KUKA KRL program: MyProgram_174().src

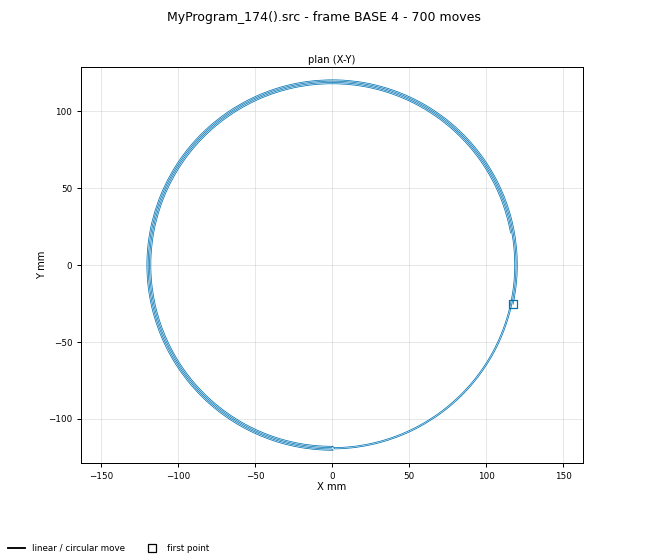
[picture p0: tool path of MyProgram_174().src in frame BASE 4, 700 of 700 moves have a stored position in this frame; points joined in program order, loops and branches not executed]
&ACCESS RVP
&REL 1
&PARAM TEMPLATE = C:\KRC\Roboter\Template\vorgabe
&PARAM EDITMASK = *
DEF MyProgram_174()
; ---- Setting reference (Base) ----
$BASE = BASE_DATA[4]

; --------------------------
; ---- Setting tool (TCP) ----
$TOOL = TOOL_DATA[3]
; --------------------------

$VEL.CP = VEL_APROX_PRINT
Startdeposition()
$VEL.CP = VEL_PRINT
LIN {X 117.5848,Y -25.4623,Z 129,A -15.6465,B 24.9508,C -1.6203,E1 25.1564,E2 461.721} C_DIS
LIN {X 118.3651,Y -21.5465,Z 129,A -14.0147,B 24.9512,C -1.6131,E1 25.1573,E2 460.1158} C_DIS
LIN {X 119.439,Y -14.4576,Z 129,A -10.3381,B 24.9498,C -1.6372,E1 25.1588,E2 456.4039} C_DIS
LIN {X 120.0869,Y -7.3562,Z 129,A -7.0535,B 24.9494,C -1.6427,E1 25.1596,E2 453.1258} C_DIS
LIN {X 120.304,Y -1.3301,Z 129,A -4.057,B 24.9485,C -1.6583,E1 25.1598,E2 450.1103} C_DIS
LIN {X 120.1794,Y 5.6204,Z 129,A -0.1852,B 24.946,C -1.6973,E1 25.1594,E2 446.1697} C_DIS
LIN {X 119.8532,Y 10.4886,Z 129,A 1.5179,B 24.9475,C -1.6737,E1 25.1591,E2 444.5324} C_DIS
LIN {X 119.0469,Y 17.3938,Z 129,A 5.2004,B 24.9457,C -1.7029,E1 25.1577,E2 440.8027} C_DIS
LIN {X 118.4357,Y 21.1537,Z 129,A 6.5409,B 24.9468,C -1.685,E1 25.1571,E2 439.5122} C_DIS
LIN {X 117.835,Y 24.2774,Z 129,A 8.2042,B 24.946,C -1.6972,E1 25.1562,E2 437.8299} C_DIS
LIN {X 116.908,Y 28.4078,Z 129,A 10.031,B 24.9462,C -1.6941,E1 25.155,E2 436.021} C_DIS
LIN {X 116.1551,Y 31.3444,Z 129,A 11.4464,B 24.946,C -1.6972,E1 25.154,E2 434.6064} C_DIS
LIN {X 115.3464,Y 34.2007,Z 129,A 12.8289,B 24.9458,C -1.7,E1 25.1529,E2 433.2252} C_DIS
LIN {X 114.4337,Y 37.1405,Z 129,A 14.334,B 24.9454,C -1.7065,E1 25.1517,E2 431.7135} C_DIS
LIN {X 113.2303,Y 40.6659,Z 129,A 16.6452,B 24.9434,C -1.7385,E1 25.1494,E2 429.3397} C_DIS
LIN {X 111.7337,Y 44.6139,Z 129,A 17.9875,B 24.9451,C -1.7113,E1 25.1482,E2 428.0691} C_DIS
LIN {X 110.031,Y 48.6627,Z 129,A 20.27,B 24.9441,C -1.7268,E1 25.1456,E2 425.7625} C_DIS
LIN {X 108.4702,Y 52.0451,Z 129,A 21.902,B 24.9442,C -1.7249,E1 25.1437,E2 424.1438} C_DIS
LIN {X 107.1163,Y 54.7776,Z 129,A 23.4021,B 24.9438,C -1.7314,E1 25.1418,E2 422.6363} C_DIS
LIN {X 105.3261,Y 58.1484,Z 129,A 25.0841,B 24.9439,C -1.7297,E1 25.1396,E2 420.9671} C_DIS
LIN {X 102.3478,Y 63.2435,Z 129,A 28.0641,B 24.9429,C -1.7456,E1 25.1353,E2 417.9649} C_DIS
LIN {X 100.5218,Y 66.105,Z 129,A 29.6094,B 24.9429,C -1.7464,E1 25.1329,E2 416.4254} C_DIS
LIN {X 98.1341,Y 69.6009,Z 129,A 31.5754,B 24.9427,C -1.7491,E1 25.1298,E2 414.4627} C_DIS
LIN {X 96.3458,Y 72.0557,Z 129,A 32.9323,B 24.9427,C -1.7484,E1 25.1276,E2 413.1141} C_DIS
LIN {X 94.6391,Y 74.2838,Z 129,A 34.2809,B 24.9425,C -1.7522,E1 25.1253,E2 411.7627} C_DIS
LIN {X 92.4033,Y 77.0464,Z 129,A 36.0716,B 24.9419,C -1.7611,E1 25.1221,E2 409.9593} C_DIS
LIN {X 89.7768,Y 80.0915,Z 129,A 37.9511,B 24.9417,C -1.7638,E1 25.1186,E2 408.0819} C_DIS
LIN {X 86.1601,Y 83.9723,Z 129,A 40.578,B 24.941,C -1.7743,E1 25.1136,E2 405.4416} C_DIS
LIN {X 83.2787,Y 86.8287,Z 129,A 43.2363,B 24.9383,C -1.8138,E1 25.1081,E2 402.701} C_DIS
LIN {X 79.152,Y 90.606,Z 129,A 45.0016,B 24.9409,C -1.7755,E1 25.1046,E2 401.0334} C_DIS
LIN {X 76.7994,Y 92.6085,Z 129,A 46.5139,B 24.9406,C -1.7803,E1 25.1013,E2 399.5155} C_DIS
LIN {X 73.8322,Y 94.9922,Z 129,A 48.3061,B 24.9404,C -1.7827,E1 25.0974,E2 397.7242} C_DIS
LIN {X 71.1983,Y 96.9809,Z 129,A 49.8066,B 24.9404,C -1.7821,E1 25.094,E2 396.2305} C_DIS
LIN {X 66.3731,Y 100.345,Z 129,A 52.681,B 24.9399,C -1.7903,E1 25.0874,E2 393.3466} C_DIS
LIN {X 63.7075,Y 102.058,Z 129,A 54.1758,B 24.9399,C -1.792,E1 25.0839,E2 391.8525} C_DIS
LIN {X 60.134,Y 104.2038,Z 129,A 56.1904,B 24.9395,C -1.7964,E1 25.079,E2 389.8338} C_DIS
LIN {X 56.8311,Y 106.0427,Z 129,A 58.0046,B 24.9393,C -1.7995,E1 25.0746,E2 388.0174} C_DIS
LIN {X 53.5539,Y 107.7333,Z 129,A 59.5541,B 24.9398,C -1.792,E1 25.0708,E2 386.4898} C_DIS
LIN {X 50.9117,Y 109.0069,Z 129,A 61.1282,B 24.9391,C -1.8021,E1 25.0667,E2 384.896} C_DIS
LIN {X 47.438,Y 110.5649,Z 129,A 62.9607,B 24.9389,C -1.8051,E1 25.0621,E2 383.0609} C_DIS
LIN {X 43.3807,Y 112.2186,Z 129,A 65.3004,B 24.938,C -1.8192,E1 25.0559,E2 380.6932} C_DIS
LIN {X 39.022,Y 113.8074,Z 129,A 67.1584,B 24.939,C -1.8046,E1 25.0511,E2 378.8734} C_DIS
LIN {X 35.8816,Y 114.8349,Z 129,A 68.9526,B 24.9382,C -1.8162,E1 25.0463,E2 377.055} C_DIS
LIN {X 31.5206,Y 116.1075,Z 129,A 70.8724,B 24.9388,C -1.8063,E1 25.0412,E2 375.1618} C_DIS
LIN {X 28.8672,Y 116.7959,Z 129,A 72.2811,B 24.9385,C -1.8119,E1 25.0373,E2 373.7419} C_DIS
LIN {X 25.2991,Y 117.6204,Z 129,A 74.3615,B 24.9373,C -1.8285,E1 25.0316,E2 371.625} C_DIS
LIN {X 21.8309,Y 118.3139,Z 129,A 75.7189,B 24.9383,C -1.814,E1 25.0279,E2 370.3036} C_DIS
LIN {X 18.5374,Y 118.8733,Z 129,A 77.239,B 24.9385,C -1.8112,E1 25.0238,E2 368.7915} C_DIS
LIN {X 15.7016,Y 119.2812,Z 129,A 78.6782,B 24.9383,C -1.815,E1 25.0198,E2 367.3445} C_DIS
LIN {X 9.3605,Y 119.9454,Z 129,A 81.6568,B 24.9384,C -1.8127,E1 25.0115,E2 364.3733} C_DIS
LIN {X 6.6678,Y 120.125,Z 129,A 83.2519,B 24.9374,C -1.827,E1 25.007,E2 362.745} C_DIS
LIN {X 2.0677,Y 120.2922,Z 129,A 85.7518,B 24.9365,C -1.8409,E1 24.9999,E2 360.2125} C_DIS
LIN {X -2.5546,Y 120.2833,Z 129,A 87.4564,B 24.9381,C -1.8174,E1 24.9953,E2 358.5634} C_DIS
LIN {X -9.7683,Y 119.9128,Z 129,A 90.5059,B 24.9394,C -1.7983,E1 24.9869,E2 355.5582} C_DIS
LIN {X -15.2296,Y 119.3423,Z 129,A 93.3875,B 24.9387,C -1.8089,E1 24.9789,E2 352.6498} C_DIS
LIN {X -18.4144,Y 118.8923,Z 129,A 95.5576,B 24.9368,C -1.8368,E1 24.9727,E2 350.4114} C_DIS
LIN {X -22.9909,Y 118.093,Z 129,A 97.1937,B 24.9387,C -1.8089,E1 24.9684,E2 348.84} C_DIS
LIN {X -26.6923,Y 117.3122,Z 129,A 98.9485,B 24.9389,C -1.8052,E1 24.9636,E2 347.0918} C_DIS
LIN {X -29.9813,Y 116.5144,Z 129,A 100.4878,B 24.9392,C -1.8004,E1 24.9594,E2 345.5618} C_DIS
LIN {X -33.4189,Y 115.5771,Z 129,A 102.3932,B 24.9387,C -1.8078,E1 24.9543,E2 343.6355} C_DIS
LIN {X -37.056,Y 114.461,Z 129,A 104.0991,B 24.9392,C -1.801,E1 24.9498,E2 341.9429} C_DIS
LIN {X -40.6481,Y 113.2369,Z 129,A 105.7919,B 24.9397,C -1.7936,E1 24.9453,E2 340.2643} C_DIS
LIN {X -46.0596,Y 111.1463,Z 129,A 108.7278,B 24.9394,C -1.7974,E1 24.9377,E2 337.313} C_DIS
LIN {X -49.0639,Y 109.8516,Z 129,A 110.2468,B 24.9397,C -1.7934,E1 24.9338,E2 335.8} C_DIS
LIN {X -54.1485,Y 107.4378,Z 129,A 112.984,B 24.9398,C -1.7916,E1 24.9269,E2 333.0599} C_DIS
LIN {X -57.1443,Y 105.8729,Z 129,A 114.6607,B 24.9398,C -1.7918,E1 24.9228,E2 331.3781} C_DIS
LIN {X -63.8759,Y 101.9528,Z 129,A 118.332,B 24.9404,C -1.7833,E1 24.914,E2 327.716} C_DIS
LIN {X -67.4437,Y 99.6284,Z 129,A 120.2451,B 24.941,C -1.7742,E1 24.9096,E2 325.818} C_DIS
LIN {X -71.7113,Y 96.6045,Z 129,A 122.8725,B 24.941,C -1.775,E1 24.9036,E2 323.1797} C_DIS
LIN {X -76.7717,Y 92.6316,Z 129,A 125.8608,B 24.9416,C -1.765,E1 24.8971,E2 320.2041} C_DIS
LIN {X -78.9489,Y 90.7833,Z 129,A 127.3315,B 24.9416,C -1.7667,E1 24.894,E2 318.7236} C_DIS
LIN {X -82.2494,Y 87.8041,Z 129,A 129.3861,B 24.942,C -1.759,E1 24.8898,E2 316.679} C_DIS
LIN {X -86.2573,Y 83.8715,Z 129,A 132.1268,B 24.9423,C -1.7553,E1 24.8843,E2 313.9355} C_DIS
LIN {X -89.1805,Y 80.7576,Z 129,A 134.1936,B 24.9425,C -1.7515,E1 24.8804,E2 311.8685} C_DIS
LIN {X -91.5631,Y 78.0428,Z 129,A 136.3235,B 24.9416,C -1.7649,E1 24.8765,E2 309.6971} C_DIS
LIN {X -94.1174,Y 74.9438,Z 129,A 137.6651,B 24.9436,C -1.735,E1 24.8743,E2 308.4205} C_DIS
LIN {X -97.8236,Y 70.0361,Z 129,A 141.1343,B 24.9426,C -1.7503,E1 24.8684,E2 304.8981} C_DIS
LIN {X -99.9834,Y 66.9195,Z 129,A 142.6448,B 24.9438,C -1.7324,E1 24.8661,E2 303.4226} C_DIS
LIN {X -102.0142,Y 63.7776,Z 129,A 144.293,B 24.9445,C -1.7216,E1 24.8637,E2 301.7919} C_DIS
LIN {X -103.3027,Y 61.671,Z 129,A 145.6708,B 24.9441,C -1.7268,E1 24.8617,E2 300.3945} C_DIS
LIN {X -106.9409,Y 55.1207,Z 129,A 148.9682,B 24.9455,C -1.7046,E1 24.8573,E2 297.1327} C_DIS
LIN {X -110.0031,Y 48.7267,Z 129,A 152.6095,B 24.9455,C -1.7056,E1 24.853,E2 293.4693} C_DIS
LIN {X -111.3647,Y 45.5238,Z 129,A 154.1469,B 24.9461,C -1.6953,E1 24.8513,E2 291.9477} C_DIS
LIN {X -112.6193,Y 42.3256,Z 129,A 157.0841,B 24.9428,C -1.7465,E1 24.8484,E2 288.872} C_DIS
LIN {X -115.0863,Y 35.0709,Z 129,A 159.0089,B 24.9483,C -1.6605,E1 24.8469,E2 287.1411} C_DIS
LIN {X -117.0482,Y 27.8334,Z 129,A 163.1341,B 24.9476,C -1.6724,E1 24.8439,E2 282.9634} C_DIS
LIN {X -117.7924,Y 24.4851,Z 129,A 164.7267,B 24.948,C -1.6654,E1 24.8429,E2 281.3782} C_DIS
LIN {X -118.3955,Y 21.3774,Z 129,A 166.2942,B 24.9482,C -1.6631,E1 24.8421,E2 279.8069} C_DIS
LIN {X -119.0397,Y 17.4443,Z 129,A 168.2482,B 24.9484,C -1.6593,E1 24.8413,E2 277.8504} C_DIS
LIN {X -119.4912,Y 14.0112,Z 129,A 169.8077,B 24.949,C -1.6501,E1 24.8407,E2 276.3035} C_DIS
LIN {X -119.8861,Y 10.1024,Z 129,A 171.7667,B 24.9491,C -1.6477,E1 24.8402,E2 274.3384} C_DIS
LIN {X -120.139,Y 6.4136,Z 129,A 173.4658,B 24.9496,C -1.6393,E1 24.84,E2 272.6491} C_DIS
LIN {X -120.28,Y 2.7339,Z 129,A 175.1714,B 24.9501,C -1.6315,E1 24.8398,E2 270.9518} C_DIS
LIN {X -120.3084,Y -0.6361,Z 129,A 176.8374,B 24.9503,C -1.6289,E1 24.8398,E2 269.2821} C_DIS
LIN {X -120.2335,Y -4.3356,Z 129,A 178.7511,B 24.9503,C -1.6296,E1 24.84,E2 267.3552} C_DIS
LIN {X -120.0348,Y -8.1312,Z 129,A -179.6085,B 24.951,C -1.6165,E1 24.8402,E2 265.7361} C_DIS
LIN {X -119.7828,Y -11.2509,Z 129,A -178.0156,B 24.951,C -1.6161,E1 24.8406,E2 264.1347} C_DIS
LIN {X -119.3925,Y -14.842,Z 129,A -176.2789,B 24.9514,C -1.6112,E1 24.8412,E2 262.3992} C_DIS
LIN {X -118.9209,Y -18.2295,Z 129,A -174.6385,B 24.9516,C -1.6065,E1 24.8418,E2 260.7603} C_DIS
LIN {X -118.257,Y -22.1389,Z 129,A -172.694,B 24.9519,C -1.6029,E1 24.8428,E2 258.8128} C_DIS
LIN {X -117.5326,Y -25.7013,Z 129,A -171.0443,B 24.9524,C -1.594,E1 24.8438,E2 257.1747} C_DIS
LIN {X -116.9844,Y -28.0949,Z 129,A -169.5097,B 24.9517,C -1.606,E1 24.8448,E2 255.6023} C_DIS
LIN {X -116.1801,Y -31.252,Z 129,A -167.2589,B 24.9501,C -1.6317,E1 24.8465,E2 253.2772} C_DIS
LIN {X -114.3114,Y -37.5184,Z 129,A -164.9234,B 24.9527,C -1.5882,E1 24.8484,E2 251.032} C_DIS
LIN {X -112.1931,Y -43.4456,Z 129,A -162.0631,B 24.9536,C -1.5733,E1 24.8512,E2 248.1912} C_DIS
LIN {X -110.8606,Y -46.7375,Z 129,A -160.4971,B 24.9542,C -1.5629,E1 24.8528,E2 246.6412} C_DIS
LIN {X -109.7148,Y -49.3674,Z 129,A -158.9868,B 24.9541,C -1.5652,E1 24.8546,E2 245.1172} C_DIS
LIN {X -107.9363,Y -53.1445,Z 129,A -157.0147,B 24.9545,C -1.5588,E1 24.8569,E2 243.1495} C_DIS
LIN {X -106.2522,Y -56.437,Z 129,A -155.3382,B 24.955,C -1.5502,E1 24.8591,E2 241.4846} C_DIS
LIN {X -103.1537,Y -61.9211,Z 129,A -152.1677,B 24.955,C -1.5494,E1 24.8635,E2 238.2994} C_DIS
LIN {X -101.2566,Y -64.9736,Z 129,A -150.6151,B 24.9557,C -1.538,E1 24.8658,E2 236.7662} C_DIS
LIN {X -98.4759,Y -69.1178,Z 129,A -148.0491,B 24.9556,C -1.5401,E1 24.8699,E2 234.1824} C_DIS
LIN {X -94.2815,Y -74.7362,Z 129,A -144.7252,B 24.9561,C -1.5312,E1 24.8755,E2 230.8638} C_DIS
LIN {X -91.7009,Y -77.881,Z 129,A -142.9284,B 24.9567,C -1.5204,E1 24.8787,E2 229.0844} C_DIS
LIN {X -86.961,Y -83.1415,Z 129,A -139.5195,B 24.957,C -1.5143,E1 24.8851,E2 225.6749} C_DIS
LIN {X -82.9842,Y -87.1125,Z 129,A -136.6202,B 24.9568,C -1.5185,E1 24.8909,E2 222.7537} C_DIS
LIN {X -79.8287,Y -90.012,Z 129,A -134.6188,B 24.9571,C -1.5126,E1 24.8951,E2 220.7582} C_DIS
LIN {X -76.4008,Y -92.9397,Z 129,A -132.5717,B 24.9576,C -1.504,E1 24.8994,E2 218.7237} C_DIS
LIN {X -73.5729,Y -95.1921,Z 129,A -131.0956,B 24.9584,C -1.49,E1 24.9026,E2 217.2755} C_DIS
LIN {X -70.5918,Y -97.4229,Z 129,A -128.601,B 24.9568,C -1.5191,E1 24.9084,E2 214.7028} C_DIS
LIN {X -67.4071,Y -99.6532,Z 129,A -127.2311,B 24.9582,C -1.4944,E1 24.9114,E2 213.3872} C_DIS
LIN {X -64.4112,Y -101.6176,Z 129,A -125.3419,B 24.9579,C -1.4999,E1 24.9159,E2 211.4787} C_DIS
LIN {X -61.2353,Y -103.5602,Z 129,A -123.7134,B 24.9584,C -1.4908,E1 24.9197,E2 209.867} C_DIS
LIN {X -57.9655,Y -105.4274,Z 129,A -121.8623,B 24.9584,C -1.4908,E1 24.9243,E2 208.0102} C_DIS
LIN {X -54.4907,Y -107.2628,Z 129,A -119.9679,B 24.9584,C -1.4895,E1 24.929,E2 206.114} C_DIS
LIN {X -50.8664,Y -109.028,Z 129,A -118.1583,B 24.9588,C -1.4822,E1 24.9335,E2 204.3171} C_DIS
LIN {X -46.2893,Y -111.0495,Z 129,A -115.4283,B 24.9581,C -1.4954,E1 24.9406,E2 201.5494} C_DIS
LIN {X -41.4285,Y -112.9522,Z 129,A -113.2356,B 24.959,C -1.4796,E1 24.9462,E2 199.3895} C_DIS
LIN {X -36.483,Y -114.6464,Z 129,A -110.7556,B 24.9591,C -1.4771,E1 24.9528,E2 196.9107} C_DIS
LIN {X -33.2199,Y -115.6335,Z 129,A -109.1067,B 24.9591,C -1.4771,E1 24.9572,E2 195.2591} C_DIS
LIN {X -30.3339,Y -116.4237,Z 129,A -107.609,B 24.959,C -1.4796,E1 24.9613,E2 193.7532} C_DIS
LIN {X -24.8979,Y -117.7076,Z 129,A -104.9009,B 24.959,C -1.4805,E1 24.9687,E2 191.0396} C_DIS
LIN {X -21.1668,Y -118.4333,Z 129,A -103.4454,B 24.9599,C -1.4635,E1 24.9726,E2 189.623} C_DIS
LIN {X -18.2676,Y -118.915,Z 129,A -101.9188,B 24.9596,C -1.4689,E1 24.9768,E2 188.082} C_DIS
LIN {X -11.8652,Y -119.7252,Z 129,A -98.4432,B 24.9586,C -1.4871,E1 24.9866,E2 184.561} C_DIS
LIN {X -6.1615,Y -120.153,Z 129,A -95.4276,B 24.9578,C -1.501,E1 24.9951,E2 181.5117} C_DIS
LIN {X -1.7022,Y -120.2989,Z 129,A -93.9382,B 24.9594,C -1.4714,E1 24.9991,E2 180.0922} C_DIS
LIN {X 0.8239,Y -120.3026,Z 129,A -91.9719,B 24.9574,C -1.5078,E1 25.0048,E2 178.0397} C_DIS
Enddeposition()
LIN {X 0.8239,Y -120.3026,Z 129,A -91.9719,B 24.9574,C -1.5078,E1 25.0048,E2 178.0397} C_DIS
Startdeposition()
$VEL.CP = VEL_PRINT
LIN {X -0.4367,Y -119.4615,Z 129,A -94.6116,B 24.9618,C -1.4278,E1 24.9969,E2 180.8689} C_DIS
LIN {X -4.7108,Y -119.3696,Z 129,A -96.1553,B 24.9606,C -1.4505,E1 24.9927,E2 182.3589} C_DIS
LIN {X -8.9928,Y -119.1241,Z 129,A -98.2312,B 24.9606,C -1.4496,E1 24.9869,E2 184.4378} C_DIS
LIN {X -12.4268,Y -118.8138,Z 129,A -100.1589,B 24.9613,C -1.4374,E1 24.9815,E2 186.3955} C_DIS
LIN {X -15.7199,Y -118.4237,Z 129,A -101.636,B 24.961,C -1.4428,E1 24.9774,E2 187.861} C_DIS
LIN {X -20.2124,Y -117.7407,Z 129,A -103.6777,B 24.9606,C -1.4497,E1 24.9718,E2 189.8882} C_DIS
LIN {X -23.8423,Y -117.0587,Z 129,A -105.3557,B 24.9604,C -1.4546,E1 24.9673,E2 191.5563} C_DIS
LIN {X -28.0159,Y -116.1308,Z 129,A -107.4362,B 24.9604,C -1.4543,E1 24.9616,E2 193.6404} C_DIS
LIN {X -31.5736,Y -115.2148,Z 129,A -109.1973,B 24.9604,C -1.4554,E1 24.9568,E2 195.4014} C_DIS
LIN {X -35.2602,Y -114.1397,Z 129,A -110.8974,B 24.9599,C -1.4631,E1 24.9523,E2 197.0862} C_DIS
LIN {X -37.9528,Y -113.2731,Z 129,A -112.4923,B 24.9604,C -1.4535,E1 24.948,E2 198.7067} C_DIS
LIN {X -41.8827,Y -111.8803,Z 129,A -114.5936,B 24.9606,C -1.4508,E1 24.9425,E2 200.8187} C_DIS
LIN {X -46.2868,Y -110.1303,Z 129,A -116.8437,B 24.9604,C -1.4542,E1 24.9367,E2 203.0659} C_DIS
LIN {X -50.2593,Y -108.3752,Z 129,A -118.7592,B 24.9599,C -1.4639,E1 24.9319,E2 204.9628} C_DIS
LIN {X -53.3538,Y -106.8861,Z 129,A -120.5285,B 24.96,C -1.4606,E1 24.9274,E2 206.7448} C_DIS
LIN {X -56.9088,Y -105.0359,Z 129,A -122.2931,B 24.9595,C -1.4701,E1 24.9231,E2 208.4917} C_DIS
LIN {X -59.5047,Y -103.5874,Z 129,A -123.7836,B 24.9595,C -1.4692,E1 24.9195,E2 209.9885} C_DIS
LIN {X -62.9285,Y -101.5447,Z 129,A -125.7339,B 24.9595,C -1.4704,E1 24.9148,E2 211.9421} C_DIS
LIN {X -65.9755,Y -99.5914,Z 129,A -127.414,B 24.9592,C -1.4756,E1 24.9109,E2 213.6152} C_DIS
LIN {X -71.648,Y -95.5914,Z 129,A -130.8507,B 24.9592,C -1.4766,E1 24.9031,E2 217.0614} C_DIS
LIN {X -75.1059,Y -92.8993,Z 129,A -132.9989,B 24.959,C -1.4785,E1 24.8983,E2 219.2131} C_DIS
LIN {X -78.417,Y -90.122,Z 129,A -134.955,B 24.9585,C -1.4876,E1 24.8942,E2 221.1552} C_DIS
LIN {X -80.9818,Y -87.8247,Z 129,A -136.5887,B 24.9583,C -1.4917,E1 24.8908,E2 222.7857} C_DIS
LIN {X -84.473,Y -84.4747,Z 129,A -139.0755,B 24.9584,C -1.4895,E1 24.8858,E2 225.2883} C_DIS
LIN {X -87.1368,Y -81.7212,Z 129,A -141.3008,B 24.9591,C -1.477,E1 24.8815,E2 227.5529} C_DIS
LIN {X -89.8475,Y -78.7312,Z 129,A -142.7343,B 24.9577,C -1.5029,E1 24.879,E2 228.9313} C_DIS
LIN {X -91.9677,Y -76.2437,Z 129,A -144.2811,B 24.9574,C -1.5075,E1 24.8762,E2 230.4743} C_DIS
LIN {X -93.5829,Y -74.2525,Z 129,A -146.3872,B 24.9593,C -1.4732,E1 24.8724,E2 232.6718} C_DIS
LIN {X -97.034,Y -69.6828,Z 129,A -148.1,B 24.9565,C -1.5239,E1 24.8697,E2 234.2722} C_DIS
LIN {X -99.5013,Y -66.1122,Z 129,A -150.4503,B 24.9568,C -1.5178,E1 24.866,E2 236.6488} C_DIS
LIN {X -101.3587,Y -63.2264,Z 129,A -152.0825,B 24.9566,C -1.5227,E1 24.8636,E2 238.2774} C_DIS
LIN {X -102.6529,Y -61.1037,Z 129,A -153.6613,B 24.9573,C -1.5096,E1 24.8613,E2 239.8957} C_DIS
LIN {X -104.4091,Y -58.0512,Z 129,A -155.2542,B 24.9568,C -1.5183,E1 24.8591,E2 241.4763} C_DIS
LIN {X -106.8872,Y -53.3516,Z 129,A -157.2967,B 24.9552,C -1.5468,E1 24.8566,E2 243.4617} C_DIS
LIN {X -107.7926,Y -51.4973,Z 129,A -158.616,B 24.9558,C -1.5356,E1 24.8549,E2 244.8147} C_DIS
LIN {X -109.4169,Y -47.9493,Z 129,A -160.3511,B 24.9552,C -1.5468,E1 24.8529,E2 246.5328} C_DIS
LIN {X -110.6429,Y -45.0478,Z 129,A -161.8964,B 24.955,C -1.5498,E1 24.8513,E2 248.0795} C_DIS
LIN {X -112.9279,Y -38.9721,Z 129,A -165.1325,B 24.9548,C -1.5539,E1 24.8482,E2 251.3242} C_DIS
LIN {X -114.0663,Y -35.497,Z 129,A -166.8077,B 24.9543,C -1.5626,E1 24.8467,E2 252.9882} C_DIS
LIN {X -115.2132,Y -31.5795,Z 129,A -169.4043,B 24.9555,C -1.542,E1 24.8448,E2 255.6491} C_DIS
LIN {X -116.3192,Y -27.2233,Z 129,A -170.9535,B 24.9536,C -1.5739,E1 24.8438,E2 257.1311} C_DIS
LIN {X -117.0179,Y -24.0408,Z 129,A -172.5595,B 24.9534,C -1.5771,E1 24.8428,E2 258.7391} C_DIS
LIN {X -117.7743,Y -20.0114,Z 129,A -174.5138,B 24.953,C -1.5838,E1 24.8419,E2 260.689} C_DIS
LIN {X -118.2819,Y -16.7494,Z 129,A -176.0889,B 24.9527,C -1.5892,E1 24.8412,E2 262.2606} C_DIS
LIN {X -118.7363,Y -13.1676,Z 129,A -177.979,B 24.9527,C -1.5881,E1 24.8406,E2 264.1645} C_DIS
LIN {X -119.0639,Y -9.7468,Z 129,A -179.5112,B 24.9521,C -1.5983,E1 24.8402,E2 265.6816} C_DIS
LIN {X -119.289,Y -6.4272,Z 129,A 178.8946,B 24.9518,C -1.6036,E1 24.84,E2 267.2728} C_DIS
LIN {X -119.4354,Y -2.54,Z 129,A 176.9999,B 24.9515,C -1.6084,E1 24.8398,E2 269.1673} C_DIS
LIN {X -119.459,Y 0.8647,Z 129,A 175.3431,B 24.9513,C -1.6128,E1 24.8398,E2 270.8238} C_DIS
LIN {X -119.3701,Y 4.7013,Z 129,A 173.4743,B 24.951,C -1.6176,E1 24.84,E2 272.6924} C_DIS
LIN {X -119.1844,Y 8.1378,Z 129,A 171.8667,B 24.9505,C -1.6248,E1 24.8402,E2 274.2924} C_DIS
LIN {X -118.8854,Y 11.7429,Z 129,A 169.9935,B 24.9505,C -1.6248,E1 24.8407,E2 276.1771} C_DIS
LIN {X -118.4752,Y 15.3227,Z 129,A 168.3806,B 24.9499,C -1.6352,E1 24.8412,E2 277.7747} C_DIS
LIN {X -117.9774,Y 18.7825,Z 129,A 166.5708,B 24.9499,C -1.6351,E1 24.842,E2 279.5955} C_DIS
LIN {X -117.3438,Y 22.3966,Z 129,A 164.9148,B 24.9493,C -1.6451,E1 24.8428,E2 281.2373} C_DIS
LIN {X -116.6098,Y 25.9531,Z 129,A 163.2229,B 24.9488,C -1.6528,E1 24.8438,E2 282.9209} C_DIS
LIN {X -115.0117,Y 32.3036,Z 129,A 159.9889,B 24.9484,C -1.659,E1 24.8461,E2 286.1591} C_DIS
LIN {X -113.8481,Y 36.1958,Z 129,A 157.1715,B 24.9503,C -1.6293,E1 24.8485,E2 289.0636} C_DIS
LIN {X -112.0446,Y 41.442,Z 129,A 155.2843,B 24.9478,C -1.6696,E1 24.8502,E2 290.8654} C_DIS
LIN {X -110.7115,Y 44.8791,Z 129,A 153.5762,B 24.9473,C -1.6776,E1 24.852,E2 292.5639} C_DIS
LIN {X -109.5996,Y 47.5304,Z 129,A 151.5129,B 24.9488,C -1.6534,E1 24.8544,E2 294.6961} C_DIS
LIN {X -107.6494,Y 51.7953,Z 129,A 149.89,B 24.9467,C -1.6862,E1 24.8562,E2 296.2497} C_DIS
LIN {X -105.9277,Y 55.2332,Z 129,A 147.9932,B 24.9465,C -1.6895,E1 24.8586,E2 298.1488} C_DIS
LIN {X -103.5203,Y 59.6214,Z 129,A 145.3426,B 24.9467,C -1.6862,E1 24.8623,E2 300.8213} C_DIS
LIN {X -101.0364,Y 63.7423,Z 129,A 143.2064,B 24.9458,C -1.7,E1 24.8654,E2 302.9355} C_DIS
LIN {X -98.2327,Y 67.982,Z 129,A 140.8781,B 24.9451,C -1.7115,E1 24.869,E2 305.248} C_DIS
LIN {X -96.3822,Y 70.5806,Z 129,A 138.9402,B 24.9459,C -1.6986,E1 24.8722,E2 307.2259} C_DIS
LIN {X -94.2532,Y 73.402,Z 129,A 137.6693,B 24.9445,C -1.721,E1 24.8743,E2 308.4496} C_DIS
LIN {X -91.033,Y 77.3574,Z 129,A 135.0344,B 24.9445,C -1.7195,E1 24.879,E2 311.1002} C_DIS
LIN {X -88.7077,Y 80.0143,Z 129,A 133.3566,B 24.9443,C -1.7245,E1 24.8821,E2 312.7736} C_DIS
LIN {X -85.5042,Y 83.4309,Z 129,A 130.8525,B 24.9446,C -1.7192,E1 24.887,E2 315.3011} C_DIS
LIN {X -81.3753,Y 87.4621,Z 129,A 128.3234,B 24.9435,C -1.7359,E1 24.892,E2 317.8009} C_DIS
LIN {X -78.2776,Y 90.2438,Z 129,A 126.2862,B 24.9433,C -1.7389,E1 24.8963,E2 319.8392} C_DIS
LIN {X -76.0959,Y 92.0906,Z 129,A 124.3675,B 24.9446,C -1.7188,E1 24.9006,E2 321.813} C_DIS
LIN {X -72.3363,Y 95.0744,Z 129,A 122.7641,B 24.9424,C -1.7533,E1 24.904,E2 323.3402} C_DIS
LIN {X -68.1659,Y 98.1048,Z 129,A 120.2546,B 24.9422,C -1.7568,E1 24.9097,E2 325.85} C_DIS
LIN {X -65.0999,Y 100.1679,Z 129,A 118.5149,B 24.9418,C -1.7617,E1 24.9137,E2 327.5839} C_DIS
LIN {X -60.6138,Y 102.9425,Z 129,A 115.3842,B 24.9432,C -1.7407,E1 24.9213,E2 330.774} C_DIS
LIN {X -57.049,Y 104.9599,Z 129,A 114.0051,B 24.9413,C -1.7692,E1 24.9245,E2 332.0893} C_DIS
LIN {X -51.6116,Y 107.7377,Z 129,A 110.9488,B 24.9413,C -1.7685,E1 24.9322,E2 335.1555} C_DIS
LIN {X -47.9493,Y 109.4169,Z 129,A 109.065,B 24.941,C -1.7735,E1 24.9369,E2 337.0318} C_DIS
LIN {X -42.8333,Y 111.5202,Z 129,A 106.5075,B 24.9405,C -1.7814,E1 24.9435,E2 339.5763} C_DIS
LIN {X -38.9198,Y 112.9462,Z 129,A 104.25,B 24.9411,C -1.7726,E1 24.9495,E2 341.8591} C_DIS
LIN {X -35.3618,Y 114.1083,Z 129,A 102.678,B 24.9403,C -1.7845,E1 24.9537,E2 343.4057} C_DIS
LIN {X -32.2489,Y 115.0273,Z 129,A 100.9668,B 24.9407,C -1.7794,E1 24.9583,E2 345.1317} C_DIS
LIN {X -28.3947,Y 116.0383,Z 129,A 99.1151,B 24.9404,C -1.7839,E1 24.9633,E2 346.9754} C_DIS
LIN {X -24.9598,Y 116.8264,Z 129,A 97.4056,B 24.9404,C -1.7846,E1 24.9679,E2 348.6854} C_DIS
LIN {X -20.1113,Y 117.7576,Z 129,A 95.052,B 24.9401,C -1.7871,E1 24.9744,E2 351.0356} C_DIS
LIN {X -17.052,Y 118.2389,Z 129,A 93.5048,B 24.9403,C -1.7854,E1 24.9787,E2 352.5883} C_DIS
LIN {X -11.5553,Y 118.9031,Z 129,A 90.8445,B 24.9402,C -1.7866,E1 24.9861,E2 355.2473} C_DIS
LIN {X -6.1538,Y 119.3041,Z 129,A 88.1952,B 24.9402,C -1.7854,E1 24.9934,E2 357.9004} C_DIS
LIN {X -2.1135,Y 119.4433,Z 129,A 86.0789,B 24.9407,C -1.7781,E1 24.9994,E2 360.0343} C_DIS
LIN {X 4.1595,Y 119.3905,Z 129,A 83.3177,B 24.94,C -1.7895,E1 25.007,E2 362.7679} C_DIS
LIN {X 7.8247,Y 119.2056,Z 129,A 81.5619,B 24.94,C -1.7897,E1 25.0119,E2 364.5226} C_DIS
LIN {X 12.7729,Y 118.7776,Z 129,A 79.0086,B 24.9405,C -1.7818,E1 25.0191,E2 367.0932} C_DIS
LIN {X 17.0048,Y 118.2456,Z 129,A 77.1012,B 24.9401,C -1.7875,E1 25.0243,E2 368.9854} C_DIS
LIN {X 20.9306,Y 117.6142,Z 129,A 75.2438,B 24.9401,C -1.7891,E1 25.0294,E2 370.8372} C_DIS
LIN {X 25.014,Y 116.8146,Z 129,A 73.2396,B 24.9401,C -1.7878,E1 25.0349,E2 372.842} C_DIS
LIN {X 28.3066,Y 116.0598,Z 129,A 71.6069,B 24.9401,C -1.7863,E1 25.0393,E2 374.4758} C_DIS
LIN {X 32.2713,Y 115.0209,Z 129,A 69.8444,B 24.9397,C -1.7943,E1 25.044,E2 376.2167} C_DIS
LIN {X 34.851,Y 114.2666,Z 129,A 68.2997,B 24.9405,C -1.7816,E1 25.0482,E2 377.7887} C_DIS
LIN {X 38.4073,Y 113.1198,Z 129,A 66.7299,B 24.9399,C -1.7903,E1 25.0523,E2 379.3348} C_DIS
LIN {X 41.7735,Y 111.9217,Z 129,A 64.8409,B 24.9406,C -1.7806,E1 25.0573,E2 381.2428} C_DIS
LIN {X 45.7752,Y 110.346,Z 129,A 62.7403,B 24.9408,C -1.7767,E1 25.0628,E2 383.3479} C_DIS
LIN {X 49.1876,Y 108.8657,Z 129,A 61.0523,B 24.9407,C -1.7792,E1 25.0671,E2 385.0259} C_DIS
LIN {X 52.7372,Y 107.1917,Z 129,A 59.179,B 24.9407,C -1.7773,E1 25.0718,E2 386.8989} C_DIS
LIN {X 55.6962,Y 105.6839,Z 129,A 57.6173,B 24.9408,C -1.7766,E1 25.0757,E2 388.4579} C_DIS
LIN {X 58.969,Y 103.8952,Z 129,A 55.7582,B 24.9412,C -1.7708,E1 25.0802,E2 390.3253} C_DIS
LIN {X 61.846,Y 102.207,Z 129,A 54.1757,B 24.9413,C -1.7692,E1 25.084,E2 391.9066} C_DIS
LIN {X 64.9082,Y 100.291,Z 129,A 52.429,B 24.9416,C -1.7658,E1 25.0881,E2 393.6558} C_DIS
LIN {X 67.515,Y 98.5561,Z 129,A 50.6854,B 24.9425,C -1.7519,E1 25.0922,E2 395.4261} C_DIS
LIN {X 71.5893,Y 95.6356,Z 129,A 48.5828,B 24.9418,C -1.7618,E1 25.0969,E2 397.4979} C_DIS
LIN {X 74.4478,Y 93.4286,Z 129,A 46.7658,B 24.9423,C -1.7546,E1 25.1009,E2 399.3252} C_DIS
LIN {X 77.4287,Y 90.9722,Z 129,A 45.0692,B 24.9421,C -1.7584,E1 25.1045,E2 401.0064} C_DIS
LIN {X 83.5476,Y 85.3889,Z 129,A 41.1962,B 24.9423,C -1.7548,E1 25.1125,E2 404.872} C_DIS
LIN {X 87.0944,Y 81.7663,Z 129,A 38.647,B 24.943,C -1.7438,E1 25.1174,E2 407.4362} C_DIS
LIN {X 89.7741,Y 78.8153,Z 129,A 36.7484,B 24.9433,C -1.7401,E1 25.1209,E2 409.3353} C_DIS
LIN {X 91.865,Y 76.3673,Z 129,A 35.3037,B 24.9432,C -1.7412,E1 25.1235,E2 410.7708} C_DIS
LIN {X 94.5274,Y 73.0462,Z 129,A 33.2033,B 24.9437,C -1.7334,E1 25.1272,E2 412.8797} C_DIS
LIN {X 96.6353,Y 70.2349,Z 129,A 31.3765,B 24.9444,C -1.7224,E1 25.1302,E2 414.7238} C_DIS
LIN {X 99.0786,Y 66.7433,Z 129,A 29.438,B 24.9444,C -1.7221,E1 25.1333,E2 416.6532} C_DIS
LIN {X 101.0866,Y 63.662,Z 129,A 27.7259,B 24.9446,C -1.72,E1 25.1359,E2 418.3619} C_DIS
LIN {X 102.526,Y 61.3185,Z 129,A 25.9649,B 24.9461,C -1.6952,E1 25.1385,E2 420.1723} C_DIS
LIN {X 104.3591,Y 58.1407,Z 129,A 24.6359,B 24.9451,C -1.711,E1 25.1402,E2 421.457} C_DIS
LIN {X 106.2039,Y 54.6995,Z 129,A 22.7666,B 24.9455,C -1.7059,E1 25.1427,E2 423.3285} C_DIS
LIN {X 107.6999,Y 51.6903,Z 129,A 21.2175,B 24.9455,C -1.7044,E1 25.1446,E2 424.8729} C_DIS
LIN {X 109.2243,Y 48.3912,Z 129,A 19.1639,B 24.9468,C -1.6843,E1 25.147,E2 426.9626} C_DIS
LIN {X 110.8373,Y 44.5701,Z 129,A 17.379,B 24.9466,C -1.6883,E1 25.1488,E2 428.7282} C_DIS
LIN {X 112.6997,Y 39.6223,Z 129,A 14.9328,B 24.9468,C -1.6851,E1 25.1512,E2 431.1685} C_DIS
LIN {X 113.9691,Y 35.8105,Z 129,A 13.037,B 24.9471,C -1.6807,E1 25.1528,E2 433.0638} C_DIS
LIN {X 114.8762,Y 32.7821,Z 129,A 11.5626,B 24.9472,C -1.6781,E1 25.154,E2 434.5361} C_DIS
LIN {X 115.6686,Y 29.8653,Z 129,A 10.0689,B 24.9476,C -1.6714,E1 25.155,E2 436.0369} C_DIS
LIN {X 116.4796,Y 26.5292,Z 129,A 8.4278,B 24.948,C -1.6665,E1 25.1561,E2 437.68} C_DIS
LIN {X 117.2536,Y 22.8656,Z 129,A 6.6651,B 24.9482,C -1.6624,E1 25.1571,E2 439.442} C_DIS
LIN {X 117.7305,Y 20.2738,Z 129,A 5.2526,B 24.9489,C -1.6512,E1 25.1578,E2 440.8728} C_DIS
LIN {X 118.587,Y 14.4419,Z 129,A 2.5537,B 24.9491,C -1.6483,E1 25.1588,E2 443.5625} C_DIS
LIN {X 118.9619,Y 10.9185,Z 129,A 1.0112,B 24.949,C -1.6505,E1 25.1592,E2 445.0908} C_DIS
LIN {X 119.2905,Y 6.4009,Z 129,A -1.5828,B 24.9506,C -1.6229,E1 25.1597,E2 447.7343} C_DIS
LIN {X 119.4287,Y 2.8979,Z 129,A -2.9779,B 24.9501,C -1.6313,E1 25.1597,E2 449.1014} C_DIS
LIN {X 119.4605,Y -0.6261,Z 129,A -4.5907,B 24.9502,C -1.6296,E1 25.1597,E2 450.7086} C_DIS
LIN {X 119.315,Y -5.9575,Z 129,A -7.1957,B 24.9509,C -1.6189,E1 25.1595,E2 453.3234} C_DIS
LIN {X 118.8893,Y -11.7027,Z 129,A -9.9649,B 24.9515,C -1.6095,E1 25.1589,E2 456.0982} C_DIS
LIN {X 118.428,Y -15.6866,Z 129,A -12.4004,B 24.9533,C -1.5783,E1 25.158,E2 458.5928} C_DIS
LIN {X 117.7147,Y -20.3678,Z 129,A -14.1101,B 24.9521,C -1.5982,E1 25.1572,E2 460.2457} C_DIS
LIN {X 117.0483,Y -23.8925,Z 129,A -15.6767,B 24.9521,C -1.6001,E1 25.1564,E2 461.7986} C_DIS
LIN {X 116.3764,Y -26.9756,Z 129,A -17.2446,B 24.9525,C -1.5925,E1 25.1554,E2 463.3753} C_DIS
LIN {X 115.4786,Y -30.5968,Z 129,A -19.0866,B 24.953,C -1.5842,E1 25.1541,E2 465.2263} C_DIS
LIN {X 114.4536,Y -34.2285,Z 129,A -20.8677,B 24.9532,C -1.5798,E1 25.1527,E2 467.0076} C_DIS
LIN {X 113.1972,Y -38.1778,Z 129,A -22.8663,B 24.9536,C -1.5729,E1 25.151,E2 469.011} C_DIS
LIN {X 111.7895,Y -42.1224,Z 129,A -24.7625,B 24.9536,C -1.5721,E1 25.1492,E2 470.8986} C_DIS
LIN {X 110.598,Y -45.1579,Z 129,A -26.3467,B 24.954,C -1.5662,E1 25.1475,E2 472.4879} C_DIS
LIN {X 109.0521,Y -48.774,Z 129,A -27.9812,B 24.9537,C -1.5727,E1 25.1458,E2 474.0982} C_DIS
LIN {X 107.215,Y -52.6902,Z 129,A -30.2935,B 24.9547,C -1.5547,E1 25.143,E2 476.4404} C_DIS
LIN {X 105.5693,Y -55.9138,Z 129,A -32.4251,B 24.9561,C -1.5303,E1 25.1401,E2 478.6182} C_DIS
LIN {X 103.7645,Y -59.1964,Z 129,A -33.8093,B 24.9553,C -1.545,E1 25.1383,E2 479.9607} C_DIS
LIN {X 100.9582,Y -63.8675,Z 129,A -36.4632,B 24.9558,C -1.5354,E1 25.1344,E2 482.6237} C_DIS
LIN {X 98.9604,Y -66.9178,Z 129,A -38.1024,B 24.9558,C -1.5358,E1 25.1319,E2 484.2539} C_DIS
LIN {X 97.5177,Y -69.0048,Z 129,A -40.0876,B 24.9581,C -1.4953,E1 25.1286,E2 486.3249} C_DIS
LIN {X 94.3866,Y -73.2289,Z 129,A -41.9461,B 24.9567,C -1.5203,E1 25.1255,E2 488.1157} C_DIS
LIN {X 91.496,Y -76.8113,Z 129,A -44.4171,B 24.9578,C -1.5017,E1 25.121,E2 490.6192} C_DIS
LIN {X 89.2285,Y -79.4326,Z 129,A -46.3174,B 24.9586,C -1.486,E1 25.1174,E2 492.548} C_DIS
LIN {X 86.0611,Y -82.8531,Z 129,A -47.8779,B 24.9571,C -1.5127,E1 25.1146,E2 494.0386} C_DIS
LIN {X 83.7201,Y -85.2185,Z 129,A -50.0233,B 24.9588,C -1.4824,E1 25.1102,E2 496.2465} C_DIS
LIN {X 80.6945,Y -88.0883,Z 129,A -51.8932,B 24.9588,C -1.4839,E1 25.1064,E2 498.1054} C_DIS
LIN {X 77.9118,Y -90.5607,Z 129,A -53.3345,B 24.9581,C -1.4962,E1 25.1034,E2 499.512} C_DIS
LIN {X 75.0923,Y -92.9103,Z 129,A -55.0065,B 24.9581,C -1.4965,E1 25.0998,E2 501.1769} C_DIS
LIN {X 70.9192,Y -96.1343,Z 129,A -57.7024,B 24.9588,C -1.483,E1 25.0938,E2 503.8948} C_DIS
LIN {X 67.2717,Y -98.7208,Z 129,A -59.7086,B 24.9587,C -1.4852,E1 25.0892,E2 505.889} C_DIS
LIN {X 60.5328,Y -102.9904,Z 129,A -63.0921,B 24.9579,C -1.4989,E1 25.0813,E2 509.2292} C_DIS
LIN {X 55.7994,Y -105.6295,Z 129,A -66.0452,B 24.9591,C -1.4773,E1 25.074,E2 512.2247} C_DIS
LIN {X 52.342,Y -107.3868,Z 129,A -68.4563,B 24.9607,C -1.4482,E1 25.0678,E2 514.6981} C_DIS
LIN {X 48.5308,Y -109.1617,Z 129,A -69.9596,B 24.9596,C -1.4692,E1 25.0641,E2 516.148} C_DIS
LIN {X 45.284,Y -110.5467,Z 129,A -71.6231,B 24.9596,C -1.4681,E1 25.0598,E2 517.8103} C_DIS
LIN {X 42.0707,Y -111.8091,Z 129,A -73.0979,B 24.9593,C -1.4744,E1 25.056,E2 519.2671} C_DIS
LIN {X 36.2985,Y -113.8149,Z 129,A -76.2641,B 24.9601,C -1.4595,E1 25.0476,E2 522.4622} C_DIS
LIN {X 32.6323,Y -114.9186,Z 129,A -78.0075,B 24.96,C -1.4618,E1 25.0429,E2 524.1972} C_DIS
LIN {X 28.99,Y -115.8931,Z 129,A -79.8847,B 24.9603,C -1.4566,E1 25.0378,E2 526.0838} C_DIS
LIN {X 25.4194,Y -116.7262,Z 129,A -81.5902,B 24.9603,C -1.4575,E1 25.0332,E2 527.785} C_DIS
LIN {X 20.9569,Y -117.6095,Z 129,A -83.9996,B 24.9609,C -1.4451,E1 25.0265,E2 530.2209} C_DIS
LIN {X 15.4106,Y -118.4638,Z 129,A -86.4146,B 24.9603,C -1.456,E1 25.0199,E2 532.6079} C_DIS
LIN {X 12.4982,Y -118.8063,Z 129,A -88.5374,B 24.9621,C -1.4223,E1 25.0138,E2 534.8091} C_DIS
LIN {X 7.5653,Y -119.2231,Z 129,A -90.14,B 24.9603,C -1.4565,E1 25.0096,E2 536.3299} C_DIS
LIN {X 1.7446,Y -119.45,Z 129,A -93.1245,B 24.9608,C -1.4468,E1 25.0012,E2 539.3367} C_DIS
LIN {X 1.7446,Y -119.45,Z 129,A -93.1245,B 24.9608,C -1.4468,E1 25.0012,E2 539.3367} C_DIS
Enddeposition()
LIN {X 0.8193,Y -118.6108,Z 129,A -93.4617,B 24.9597,C -1.4666,E1 25.0004,E2 539.627} C_DIS
Startdeposition()
$VEL.CP = VEL_PRINT
LIN {X 4.1826,Y -118.5414,Z 129,A -90.9638,B 24.9574,C -1.5072,E1 25.0076,E2 537.0335} C_DIS
LIN {X 7.3853,Y -118.3854,Z 129,A -89.5129,B 24.9577,C -1.5032,E1 25.0116,E2 535.5924} C_DIS
LIN {X 12.0231,Y -118.0035,Z 129,A -87.4079,B 24.958,C -1.4978,E1 25.0174,E2 533.5015} C_DIS
LIN {X 15.3204,Y -117.6204,Z 129,A -85.7262,B 24.9577,C -1.5025,E1 25.0221,E2 531.8101} C_DIS
LIN {X 18.6646,Y -117.1375,Z 129,A -83.7353,B 24.9567,C -1.5204,E1 25.0277,E2 529.7786} C_DIS
LIN {X 21.9525,Y -116.5658,Z 129,A -82.5812,B 24.9578,C -1.5003,E1 25.0308,E2 528.6734} C_DIS
LIN {X 24.4445,Y -116.0694,Z 129,A -81.2199,B 24.9574,C -1.5076,E1 25.0345,E2 527.2965} C_DIS
LIN {X 27.9179,Y -115.2818,Z 129,A -79.5222,B 24.9574,C -1.5083,E1 25.0391,E2 525.5996} C_DIS
LIN {X 30.9241,Y -114.5119,Z 129,A -78.0584,B 24.9574,C -1.5083,E1 25.0431,E2 524.1382} C_DIS
LIN {X 34.3845,Y -113.5228,Z 129,A -76.2046,B 24.957,C -1.5156,E1 25.0481,E2 522.2702} C_DIS
LIN {X 39.1081,Y -111.9815,Z 129,A -74.1386,B 24.9577,C -1.5029,E1 25.0535,E2 520.2383} C_DIS
LIN {X 42.0408,Y -110.9137,Z 129,A -72.4377,B 24.9571,C -1.514,E1 25.058,E2 518.5145} C_DIS
LIN {X 45.4847,Y -109.5482,Z 129,A -70.5036,B 24.9565,C -1.5235,E1 25.063,E2 516.5626} C_DIS
LIN {X 48.8644,Y -108.0813,Z 129,A -68.8477,B 24.9567,C -1.5203,E1 25.0672,E2 514.9181} C_DIS
LIN {X 52.6418,Y -106.2925,Z 129,A -66.8591,B 24.9566,C -1.5222,E1 25.0722,E2 512.9303} C_DIS
LIN {X 55.7558,Y -104.6941,Z 129,A -64.9869,B 24.9559,C -1.5338,E1 25.0769,E2 511.036} C_DIS
LIN {X 59.1528,Y -102.8116,Z 129,A -63.3298,B 24.9563,C -1.5267,E1 25.0809,E2 509.4006} C_DIS
LIN {X 62.1074,Y -101.0558,Z 129,A -61.3225,B 24.9552,C -1.5465,E1 25.0858,E2 507.3528} C_DIS
LIN {X 66.2431,Y -98.3931,Z 129,A -59.2375,B 24.9557,C -1.5372,E1 25.0906,E2 505.2965} C_DIS
LIN {X 69.1523,Y -96.3708,Z 129,A -57.5968,B 24.9557,C -1.5374,E1 25.0943,E2 503.6613} C_DIS
LIN {X 71.9229,Y -94.3224,Z 129,A -55.9409,B 24.9555,C -1.5405,E1 25.098,E2 502.0038} C_DIS
LIN {X 74.5558,Y -92.2536,Z 129,A -54.2824,B 24.9552,C -1.5461,E1 25.1016,E2 500.3383} C_DIS
LIN {X 77.3069,Y -89.962,Z 129,A -52.5023,B 24.9548,C -1.5525,E1 25.1054,E2 498.5501} C_DIS
LIN {X 80.6845,Y -86.9467,Z 129,A -50.274,B 24.9544,C -1.5597,E1 25.11,E2 496.3138} C_DIS
LIN {X 83.2266,Y -84.5141,Z 129,A -48.716,B 24.9546,C -1.557,E1 25.1131,E2 494.7687} C_DIS
LIN {X 85.5552,Y -82.1561,Z 129,A -47.0878,B 24.9543,C -1.5623,E1 25.1163,E2 493.1348} C_DIS
LIN {X 88.9632,Y -78.4547,Z 129,A -44.6644,B 24.9539,C -1.5682,E1 25.1209,E2 490.7082} C_DIS
LIN {X 90.9485,Y -76.1434,Z 129,A -43.183,B 24.9537,C -1.5726,E1 25.1235,E2 489.2233} C_DIS
LIN {X 93.1338,Y -73.4532,Z 129,A -41.5422,B 24.9535,C -1.5755,E1 25.1264,E2 487.5833} C_DIS
LIN {X 96.2908,Y -69.2644,Z 129,A -39.0311,B 24.9531,C -1.5814,E1 25.1306,E2 485.0704} C_DIS
LIN {X 98.3233,Y -66.3462,Z 129,A -37.3633,B 24.953,C -1.5838,E1 25.1332,E2 483.4051} C_DIS
LIN {X 100.3374,Y -63.2607,Z 129,A -35.4456,B 24.9523,C -1.5957,E1 25.1361,E2 481.4691} C_DIS
LIN {X 102.2328,Y -60.1479,Z 129,A -33.9059,B 24.9526,C -1.59,E1 25.1383,E2 479.9506} C_DIS
LIN {X 103.9616,Y -57.1109,Z 129,A -31.9908,B 24.9517,C -1.6061,E1 25.1409,E2 478.0075} C_DIS
LIN {X 105.9358,Y -53.3606,Z 129,A -29.8229,B 24.9509,C -1.6183,E1 25.1437,E2 475.8225} C_DIS
LIN {X 108.1415,Y -48.7307,Z 129,A -27.6686,B 24.9514,C -1.61,E1 25.1462,E2 473.6993} C_DIS
LIN {X 109.4996,Y -45.6,Z 129,A -26.0629,B 24.9512,C -1.613,E1 25.148,E2 472.0954} C_DIS
LIN {X 110.945,Y -41.958,Z 129,A -24.1517,B 24.9508,C -1.6198,E1 25.1499,E2 470.1787} C_DIS
LIN {X 112.2409,Y -38.36,Z 129,A -22.2224,B 24.9502,C -1.6297,E1 25.1517,E2 468.237} C_DIS
LIN {X 113.3953,Y -34.7979,Z 129,A -20.3909,B 24.9498,C -1.6366,E1 25.1532,E2 466.3997} C_DIS
LIN {X 114.498,Y -30.9754,Z 129,A -18.6016,B 24.9498,C -1.6362,E1 25.1546,E2 464.6214} C_DIS
LIN {X 115.2567,Y -28.0209,Z 129,A -17.1617,B 24.9496,C -1.6394,E1 25.1555,E2 463.1825} C_DIS
LIN {X 116.0286,Y -24.6385,Z 129,A -15.3733,B 24.949,C -1.6503,E1 25.1566,E2 461.3787} C_DIS
LIN {X 116.7673,Y -20.8492,Z 129,A -13.6384,B 24.949,C -1.65,E1 25.1575,E2 459.6546} C_DIS
LIN {X 117.4179,Y -16.8025,Z 129,A -11.6899,B 24.9487,C -1.6549,E1 25.1583,E2 457.706} C_DIS
LIN {X 117.8228,Y -13.6771,Z 129,A -10.1797,B 24.9484,C -1.6593,E1 25.1588,E2 456.1944} C_DIS
LIN {X 118.189,Y -10.0489,Z 129,A -8.2416,B 24.9475,C -1.6738,E1 25.1593,E2 454.2337} C_DIS
LIN {X 118.4784,Y -5.7015,Z 129,A -6.14,B 24.9471,C -1.6805,E1 25.1597,E2 452.1287} C_DIS
LIN {X 118.5914,Y -2.3172,Z 129,A -4.6768,B 24.9473,C -1.6774,E1 25.1597,E2 450.6815} C_DIS
LIN {X 118.6109,Y 0.8732,Z 129,A -3.105,B 24.9469,C -1.684,E1 25.1597,E2 449.1036} C_DIS
LIN {X 118.5085,Y 5.0003,Z 129,A -1.0941,B 24.9464,C -1.6913,E1 25.1596,E2 447.0874} C_DIS
LIN {X 118.29,Y 8.7862,Z 129,A 0.7853,B 24.9459,C -1.6996,E1 25.1592,E2 445.1996} C_DIS
LIN {X 117.9597,Y 12.4414,Z 129,A 2.3724,B 24.9461,C -1.6962,E1 25.1588,E2 443.6299} C_DIS
LIN {X 117.534,Y 15.9841,Z 129,A 4.2951,B 24.9451,C -1.7115,E1 25.1581,E2 441.6824} C_DIS
LIN {X 117.0009,Y 19.4949,Z 129,A 5.8353,B 24.9453,C -1.7084,E1 25.1574,E2 440.1586} C_DIS
LIN {X 116.3797,Y 22.9192,Z 129,A 7.5493,B 24.9449,C -1.7153,E1 25.1565,E2 438.4383} C_DIS
LIN {X 115.5597,Y 26.7438,Z 129,A 9.3285,B 24.9449,C -1.7159,E1 25.1554,E2 436.6681} C_DIS
LIN {X 114.8405,Y 29.6809,Z 129,A 10.8083,B 24.9445,C -1.7214,E1 25.1544,E2 435.1839} C_DIS
LIN {X 113.9226,Y 33.0369,Z 129,A 12.5511,B 24.9439,C -1.7296,E1 25.1531,E2 433.4318} C_DIS
LIN {X 112.8663,Y 36.4757,Z 129,A 14.2564,B 24.9437,C -1.7334,E1 25.1517,E2 431.7272} C_DIS
LIN {X 111.4795,Y 40.5167,Z 129,A 16.7246,B 24.942,C -1.7594,E1 25.1493,E2 429.2116} C_DIS
LIN {X 110.0926,Y 44.1503,Z 129,A 18.0886,B 24.9433,C -1.7398,E1 25.148,E2 427.9013} C_DIS
LIN {X 108.6572,Y 47.5701,Z 129,A 19.929,B 24.9428,C -1.7474,E1 25.1459,E2 426.053} C_DIS
LIN {X 107.0939,Y 50.9934,Z 129,A 21.7741,B 24.9423,C -1.7539,E1 25.1437,E2 424.2024} C_DIS
LIN {X 105.5543,Y 54.1071,Z 129,A 23.3719,B 24.9423,C -1.7548,E1 25.1417,E2 422.6111} C_DIS
LIN {X 103.8282,Y 57.3522,Z 129,A 25.3195,B 24.9414,C -1.7681,E1 25.1391,E2 420.6424} C_DIS
LIN {X 102.138,Y 60.3083,Z 129,A 26.7888,B 24.9417,C -1.7641,E1 25.1371,E2 419.1901} C_DIS
LIN {X 100.3541,Y 63.234,Z 129,A 28.4003,B 24.9415,C -1.7663,E1 25.1347,E2 417.5814} C_DIS
LIN {X 98.5407,Y 66.0251,Z 129,A 30.0725,B 24.941,C -1.7736,E1 25.1321,E2 415.9003} C_DIS
LIN {X 96.6369,Y 68.7793,Z 129,A 31.66,B 24.9409,C -1.7764,E1 25.1296,E2 414.3142} C_DIS
LIN {X 94.7585,Y 71.345,Z 129,A 33.1382,B 24.9408,C -1.7774,E1 25.1271,E2 412.8405} C_DIS
LIN {X 92.3701,Y 74.412,Z 129,A 35.0851,B 24.9403,C -1.7853,E1 25.1237,E2 410.8841} C_DIS
LIN {X 90.2547,Y 76.9634,Z 129,A 36.5773,B 24.9403,C -1.7839,E1 25.1211,E2 409.4021} C_DIS
LIN {X 88.2706,Y 79.2312,Z 129,A 38.0409,B 24.9401,C -1.7877,E1 25.1184,E2 407.9362} C_DIS
LIN {X 86.0277,Y 81.6628,Z 129,A 39.9087,B 24.939,C -1.8041,E1 25.1147,E2 406.0376} C_DIS
LIN {X 83.5209,Y 84.2234,Z 129,A 41.4033,B 24.9395,C -1.7966,E1 25.1118,E2 404.5672} C_DIS
LIN {X 81.1077,Y 86.5497,Z 129,A 43.5838,B 24.9374,C -1.8269,E1 25.1073,E2 402.3241} C_DIS
LIN {X 77.8802,Y 89.4649,Z 129,A 44.9924,B 24.9394,C -1.798,E1 25.1045,E2 400.9892} C_DIS
LIN {X 75.7462,Y 91.2786,Z 129,A 46.4064,B 24.939,C -1.8036,E1 25.1014,E2 399.5676} C_DIS
LIN {X 73.4219,Y 93.1585,Z 129,A 47.8617,B 24.9388,C -1.8068,E1 25.0982,E2 398.1101} C_DIS
LIN {X 70.374,Y 95.4825,Z 129,A 49.8528,B 24.9381,C -1.8167,E1 25.0937,E2 396.1026} C_DIS
LIN {X 67.6083,Y 97.4597,Z 129,A 51.4455,B 24.9381,C -1.8172,E1 25.0901,E2 394.5143} C_DIS
LIN {X 64.2388,Y 99.713,Z 129,A 53.3136,B 24.9381,C -1.8162,E1 25.0858,E2 392.6549} C_DIS
LIN {X 61.0355,Y 101.7073,Z 129,A 55.275,B 24.9375,C -1.8255,E1 25.0811,E2 390.6777} C_DIS
LIN {X 57.5551,Y 103.7149,Z 129,A 57.0063,B 24.938,C -1.8185,E1 25.0769,E2 388.9681} C_DIS
LIN {X 54.6923,Y 105.2542,Z 129,A 58.7457,B 24.9373,C -1.8285,E1 25.0726,E2 387.21} C_DIS
LIN {X 51.2843,Y 106.9541,Z 129,A 60.4465,B 24.9376,C -1.8243,E1 25.0683,E2 385.5235} C_DIS
LIN {X 48.1352,Y 108.4099,Z 129,A 62.2106,B 24.9372,C -1.8303,E1 25.0638,E2 383.7495} C_DIS
LIN {X 44.7569,Y 109.8458,Z 129,A 63.8847,B 24.9374,C -1.8277,E1 25.0595,E2 382.0856} C_DIS
LIN {X 41.4009,Y 111.156,Z 129,A 65.7293,B 24.9369,C -1.8342,E1 25.0547,E2 380.2296} C_DIS
LIN {X 37.7768,Y 112.4375,Z 129,A 67.514,B 24.9371,C -1.8325,E1 25.05,E2 378.4524} C_DIS
LIN {X 33.1074,Y 113.9017,Z 129,A 69.7671,B 24.9373,C -1.8292,E1 25.044,E2 376.2112} C_DIS
LIN {X 28.7014,Y 115.0907,Z 129,A 72.1636,B 24.9366,C -1.8394,E1 25.0375,E2 373.7941} C_DIS
LIN {X 25.2542,Y 115.8943,Z 129,A 73.8124,B 24.9367,C -1.8375,E1 25.033,E2 372.152} C_DIS
LIN {X 21.9828,Y 116.56,Z 129,A 75.3464,B 24.9369,C -1.8346,E1 25.0288,E2 370.6267} C_DIS
LIN {X 18.5434,Y 117.1562,Z 129,A 77.0863,B 24.9367,C -1.8377,E1 25.024,E2 368.8814} C_DIS
LIN {X 15.129,Y 117.6452,Z 129,A 78.7105,B 24.9368,C -1.8362,E1 25.0195,E2 367.2621} C_DIS
LIN {X 11.8301,Y 118.0237,Z 129,A 80.2797,B 24.9368,C -1.8348,E1 25.0152,E2 365.6972} C_DIS
LIN {X 9.2808,Y 118.2504,Z 129,A 81.6183,B 24.9366,C -1.8396,E1 25.0114,E2 364.3481} C_DIS
LIN {X 4.9925,Y 118.5089,Z 129,A 83.6071,B 24.9368,C -1.8356,E1 25.0059,E2 362.3693} C_DIS
LIN {X 1.9365,Y 118.5984,Z 129,A 85.2138,B 24.9365,C -1.8413,E1 25.0014,E2 360.7495} C_DIS
LIN {X -2.2681,Y 118.5923,Z 129,A 87.142,B 24.9368,C -1.8362,E1 24.996,E2 358.8333} C_DIS
LIN {X -5.6323,Y 118.4814,Z 129,A 88.8902,B 24.9365,C -1.8411,E1 24.9911,E2 357.0731} C_DIS
LIN {X -10.0384,Y 118.1899,Z 129,A 91.0271,B 24.9365,C -1.8403,E1 24.9852,E2 354.9371} C_DIS
LIN {X -14.7549,Y 117.6937,Z 129,A 93.2402,B 24.9368,C -1.8356,E1 24.9791,E2 352.7338} C_DIS
LIN {X -18.0836,Y 117.2273,Z 129,A 94.9023,B 24.9368,C -1.8362,E1 24.9745,E2 351.0689} C_DIS
LIN {X -21.8698,Y 116.5817,Z 129,A 96.8236,B 24.9367,C -1.8377,E1 24.9692,E2 349.1421} C_DIS
LIN {X -25.8853,Y 115.7567,Z 129,A 98.793,B 24.9369,C -1.8355,E1 24.9638,E2 347.1756} C_DIS
LIN {X -29.6654,Y 114.8445,Z 129,A 100.5525,B 24.9373,C -1.8284,E1 24.9591,E2 345.4304} C_DIS
LIN {X -33.0909,Y 113.9066,Z 129,A 102.4912,B 24.9368,C -1.8364,E1 24.9538,E2 343.4697} C_DIS
LIN {X -36.6981,Y 112.7943,Z 129,A 104.106,B 24.9376,C -1.8251,E1 24.9496,E2 341.8788} C_DIS
LIN {X -41.3034,Y 111.1926,Z 129,A 106.5688,B 24.9375,C -1.8267,E1 24.9431,E2 339.4072} C_DIS
LIN {X -45.9799,Y 109.3395,Z 129,A 108.5774,B 24.9389,C -1.805,E1 24.938,E2 337.4459} C_DIS
LIN {X -49.5072,Y 107.7899,Z 129,A 110.8221,B 24.938,C -1.8188,E1 24.9322,E2 335.1628} C_DIS
LIN {X -52.7079,Y 106.2598,Z 129,A 112.7537,B 24.9375,C -1.8256,E1 24.9273,E2 333.2102} C_DIS
LIN {X -55.791,Y 104.6756,Z 129,A 114.2797,B 24.9382,C -1.8162,E1 24.9236,E2 331.7022} C_DIS
LIN {X -59.0137,Y 102.8915,Z 129,A 116.8832,B 24.9359,C -1.849,E1 24.9171,E2 329.0129} C_DIS
LIN {X -64.0563,Y 99.8301,Z 129,A 118.6473,B 24.9395,C -1.7964,E1 24.9132,E2 327.3684} C_DIS
LIN {X -66.3148,Y 98.3446,Z 129,A 120.1316,B 24.9392,C -1.8015,E1 24.9097,E2 325.8671} C_DIS
LIN {X -69.6505,Y 96.0122,Z 129,A 122.1202,B 24.9394,C -1.7984,E1 24.9052,E2 323.879} C_DIS
LIN {X -72.3027,Y 94.0298,Z 129,A 123.7019,B 24.9397,C -1.7942,E1 24.9016,E2 322.3015} C_DIS
LIN {X -75.8627,Y 91.1818,Z 129,A 125.8998,B 24.94,C -1.7892,E1 24.8969,E2 320.1073} C_DIS
LIN {X -78.4493,Y 88.9679,Z 129,A 127.8156,B 24.9395,C -1.797,E1 24.8928,E2 318.1654} C_DIS
LIN {X -81.1817,Y 86.48,Z 129,A 130.1239,B 24.9382,C -1.8153,E1 24.888,E2 315.804} C_DIS
LIN {X -84.8972,Y 82.8387,Z 129,A 131.8506,B 24.9409,C -1.7753,E1 24.8848,E2 314.1652} C_DIS
LIN {X -86.9399,Y 80.6919,Z 129,A 133.5494,B 24.9404,C -1.7831,E1 24.8815,E2 312.4404} C_DIS
LIN {X -89.9601,Y 77.3091,Z 129,A 136.1574,B 24.9396,C -1.7953,E1 24.8767,E2 309.7916} C_DIS
LIN {X -92.8059,Y 73.8681,Z 129,A 137.6041,B 24.942,C -1.7593,E1 24.8743,E2 308.424} C_DIS
LIN {X -95.064,Y 70.9383,Z 129,A 139.5533,B 24.9419,C -1.7613,E1 24.8709,E2 306.4607} C_DIS
LIN {X -97.3723,Y 67.734,Z 129,A 141.4622,B 24.9422,C -1.756,E1 24.8679,E2 304.5549} C_DIS
LIN {X -99.4946,Y 64.579,Z 129,A 143.1718,B 24.9429,C -1.7454,E1 24.8652,E2 302.862} C_DIS
LIN {X -100.9678,Y 62.2515,Z 129,A 144.8832,B 24.9421,C -1.7577,E1 24.8627,E2 301.1127} C_DIS
LIN {X -102.9089,Y 58.9833,Z 129,A 146.4685,B 24.9431,C -1.7417,E1 24.8605,E2 299.5571} C_DIS
LIN {X -104.7417,Y 55.6654,Z 129,A 148.3213,B 24.9434,C -1.7372,E1 24.858,E2 297.7052} C_DIS
LIN {X -106.3258,Y 52.5747,Z 129,A 149.9444,B 24.9439,C -1.7299,E1 24.856,E2 296.091} C_DIS
LIN {X -107.8007,Y 49.484,Z 129,A 151.9088,B 24.9434,C -1.7379,E1 24.8536,E2 294.0967} C_DIS
LIN {X -109.5943,Y 45.3745,Z 129,A 153.9619,B 24.9441,C -1.7264,E1 24.8514,E2 292.0596} C_DIS
LIN {X -111.0032,Y 41.8043,Z 129,A 155.7017,B 24.9448,C -1.7159,E1 24.8497,E2 290.3352} C_DIS
LIN {X -112.5161,Y 37.5436,Z 129,A 157.8436,B 24.9454,C -1.7072,E1 24.8477,E2 288.2017} C_DIS
LIN {X -113.3701,Y 34.879,Z 129,A 159.2073,B 24.9456,C -1.7034,E1 24.8466,E2 286.8392} C_DIS
LIN {X -114.1534,Y 32.2222,Z 129,A 160.6214,B 24.9456,C -1.7024,E1 24.8455,E2 285.4195} C_DIS
LIN {X -115.0598,Y 28.8274,Z 129,A 162.5849,B 24.9453,C -1.7081,E1 24.8441,E2 283.4309} C_DIS
LIN {X -116.1008,Y 24.2915,Z 129,A 164.6506,B 24.9463,C -1.6931,E1 24.8429,E2 281.3887} C_DIS
LIN {X -116.7581,Y 20.9001,Z 129,A 166.3257,B 24.9466,C -1.688,E1 24.8421,E2 279.7159} C_DIS
LIN {X -117.3935,Y 16.9739,Z 129,A 168.2588,B 24.947,C -1.6822,E1 24.8413,E2 277.785} C_DIS
LIN {X -117.8639,Y 13.3261,Z 129,A 170.0435,B 24.9473,C -1.6768,E1 24.8407,E2 276.0027} C_DIS
LIN {X -118.2284,Y 9.5568,Z 129,A 171.8167,B 24.9478,C -1.6685,E1 24.8402,E2 274.2387} C_DIS
LIN {X -118.4397,Y 6.4286,Z 129,A 173.3542,B 24.9481,C -1.6645,E1 24.84,E2 272.7015} C_DIS
LIN {X -118.5818,Y 2.8375,Z 129,A 175.2117,B 24.9481,C -1.6639,E1 24.8398,E2 270.8342} C_DIS
LIN {X -118.6128,Y -0.5816,Z 129,A 176.7722,B 24.9487,C -1.6547,E1 24.8398,E2 269.2863} C_DIS
LIN {X -118.5396,Y -4.2425,Z 129,A 178.6736,B 24.9487,C -1.6545,E1 24.84,E2 267.3739} C_DIS
LIN {X -118.3328,Y -8.1632,Z 129,A -179.6281,B 24.9496,C -1.64,E1 24.8402,E2 265.6998} C_DIS
LIN {X -118.0751,Y -11.3003,Z 129,A -177.9054,B 24.9494,C -1.6436,E1 24.8407,E2 263.9583} C_DIS
LIN {X -117.6331,Y -15.2223,Z 129,A -176.114,B 24.9501,C -1.6326,E1 24.8413,E2 262.1823} C_DIS
LIN {X -117.1797,Y -18.3917,Z 129,A -174.537,B 24.9503,C -1.6289,E1 24.8419,E2 260.6046} C_DIS
LIN {X -116.5195,Y -22.193,Z 129,A -172.5967,B 24.9504,C -1.6262,E1 24.8429,E2 258.6593} C_DIS
LIN {X -115.6702,Y -26.2653,Z 129,A -170.1345,B 24.9497,C -1.6391,E1 24.8444,E2 256.1519} C_DIS
LIN {X -114.7315,Y -30.1024,Z 129,A -168.7984,B 24.9515,C -1.6089,E1 24.8453,E2 254.88} C_DIS
LIN {X -114.0387,Y -32.6271,Z 129,A -167.5025,B 24.9517,C -1.6064,E1 24.8463,E2 253.5827} C_DIS
LIN {X -113.2381,Y -35.3048,Z 129,A -166.1238,B 24.9518,C -1.6034,E1 24.8474,E2 252.203} C_DIS
LIN {X -112.1936,Y -38.5003,Z 129,A -164.3662,B 24.9518,C -1.6042,E1 24.849,E2 250.4336} C_DIS
LIN {X -110.6893,Y -42.6332,Z 129,A -162.3598,B 24.9525,C -1.5928,E1 24.8509,E2 248.4429} C_DIS
LIN {X -109.526,Y -45.5374,Z 129,A -160.71,B 24.9524,C -1.5943,E1 24.8527,E2 246.7806} C_DIS
LIN {X -108.0512,Y -48.931,Z 129,A -158.9983,B 24.9529,C -1.5859,E1 24.8546,E2 245.0794} C_DIS
LIN {X -105.8371,Y -53.5537,Z 129,A -155.1229,B 24.9496,C -1.6393,E1 24.8597,E2 241.0559} C_DIS
LIN {X -102.0276,Y -60.4952,Z 129,A -152.8895,B 24.9544,C -1.5601,E1 24.8625,E2 238.9996} C_DIS
LIN {X -100.6076,Y -62.8281,Z 129,A -151.3476,B 24.954,C -1.566,E1 24.8648,E2 237.4357} C_DIS
LIN {X -98.5978,Y -65.9408,Z 129,A -149.315,B 24.9537,C -1.5718,E1 24.868,E2 235.3791} C_DIS
LIN {X -96.7471,Y -68.6248,Z 129,A -147.9039,B 24.9544,C -1.5607,E1 24.8702,E2 233.9874} C_DIS
LIN {X -94.6219,Y -71.5268,Z 129,A -145.9018,B 24.9539,C -1.5678,E1 24.8736,E2 231.9588} C_DIS
LIN {X -92.2295,Y -74.5855,Z 129,A -144.3238,B 24.955,C -1.5504,E1 24.8763,E2 230.4148} C_DIS
LIN {X -90.1645,Y -77.0692,Z 129,A -142.7448,B 24.9551,C -1.5476,E1 24.8791,E2 228.8354} C_DIS
LIN {X -87.3653,Y -80.2283,Z 129,A -140.7717,B 24.9556,C -1.5401,E1 24.8828,E2 226.8713} C_DIS
LIN {X -85.4232,Y -82.293,Z 129,A -139.333,B 24.9556,C -1.5401,E1 24.8856,E2 225.4264} C_DIS
LIN {X -82.8624,Y -84.8739,Z 129,A -137.3157,B 24.9551,C -1.5476,E1 24.8896,E2 223.3826} C_DIS
LIN {X -79.4201,Y -88.1016,Z 129,A -135.1955,B 24.9558,C -1.536,E1 24.894,E2 221.2814} C_DIS
LIN {X -76.6843,Y -90.4924,Z 129,A -133.5063,B 24.9562,C -1.5297,E1 24.8975,E2 219.6006} C_DIS
LIN {X -72.6596,Y -93.7548,Z 129,A -131.2067,B 24.9569,C -1.5162,E1 24.9025,E2 217.3247} C_DIS
LIN {X -67.3399,Y -97.6463,Z 129,A -128.04,B 24.9573,C -1.5098,E1 24.9096,E2 214.162} C_DIS
LIN {X -63.9293,Y -99.9116,Z 129,A -125.8052,B 24.9568,C -1.5179,E1 24.9149,E2 211.9007} C_DIS
LIN {X -60.9634,Y -101.7508,Z 129,A -123.9947,B 24.9567,C -1.5209,E1 24.9192,E2 210.0775} C_DIS
LIN {X -57.8261,Y -103.5635,Z 129,A -122.3829,B 24.9572,C -1.5123,E1 24.9231,E2 208.4814} C_DIS
LIN {X -54.6689,Y -105.2665,Z 129,A -120.548,B 24.957,C -1.5145,E1 24.9277,E2 206.6361} C_DIS
LIN {X -51.3858,Y -106.9054,Z 129,A -118.8373,B 24.9573,C -1.5096,E1 24.9319,E2 204.9326} C_DIS
LIN {X -47.955,Y -108.4894,Z 129,A -116.9172,B 24.9572,C -1.5117,E1 24.9369,E2 203.0028} C_DIS
LIN {X -44.6119,Y -109.9048,Z 129,A -115.229,B 24.9575,C -1.507,E1 24.9412,E2 201.322} C_DIS
LIN {X -40.7224,Y -111.4045,Z 129,A -113.2275,B 24.9575,C -1.5046,E1 24.9464,E2 199.3221} C_DIS
LIN {X -35.9943,Y -113.022,Z 129,A -110.882,B 24.9579,C -1.4995,E1 24.9526,E2 196.9842} C_DIS
LIN {X -32.9429,Y -113.9492,Z 129,A -109.1714,B 24.9575,C -1.5061,E1 24.9572,E2 195.2552} C_DIS
LIN {X -29.3301,Y -114.9306,Z 129,A -107.4843,B 24.9579,C -1.4995,E1 24.9618,E2 193.5812} C_DIS
LIN {X -25.9943,Y -115.7328,Z 129,A -105.8528,B 24.9579,C -1.4975,E1 24.9662,E2 191.9524} C_DIS
LIN {X -23.1939,Y -116.3261,Z 129,A -104.4067,B 24.9579,C -1.4997,E1 24.9702,E2 190.4991} C_DIS
LIN {X -19.862,Y -116.9395,Z 129,A -102.7836,B 24.9579,C -1.4986,E1 24.9746,E2 188.8772} C_DIS
LIN {X -16.4504,Y -117.4679,Z 129,A -101.0505,B 24.9578,C -1.5012,E1 24.9794,E2 187.1365} C_DIS
LIN {X -12.242,Y -117.9805,Z 129,A -99.1046,B 24.9581,C -1.4962,E1 24.9848,E2 185.201} C_DIS
LIN {X -9.3206,Y -118.2472,Z 129,A -97.6974,B 24.9581,C -1.4957,E1 24.9887,E2 183.7944} C_DIS
LIN {X -5.8583,Y -118.4712,Z 129,A -95.7229,B 24.9573,C -1.5095,E1 24.9943,E2 181.7866} C_DIS
LIN {X -0.832,Y -118.6111,Z 129,A -93.5378,B 24.9579,C -1.4987,E1 25.0003,E2 179.627} C_DIS
LIN {X -0.832,Y -118.6111,Z 129,A -93.5378,B 24.9579,C -1.4987,E1 25.0003,E2 179.627} C_DIS
Enddeposition()
LIN {X 0.808,Y -117.7629,Z 129,A -92.8151,B 24.9573,C -1.5104,E1 25.0025,E2 178.8767} C_DIS
Startdeposition()
$VEL.CP = VEL_PRINT
LIN {X -2.1665,Y -117.746,Z 129,A -94.9091,B 24.9589,C -1.4807,E1 24.9964,E2 181.0411} C_DIS
LIN {X -5.1286,Y -117.6542,Z 129,A -96.3512,B 24.9589,C -1.4805,E1 24.9924,E2 182.4838} C_DIS
LIN {X -8.0018,Y -117.4938,Z 129,A -97.7824,B 24.959,C -1.4791,E1 24.9884,E2 183.919} C_DIS
LIN {X -11.5444,Y -117.201,Z 129,A -99.4943,B 24.959,C -1.4799,E1 24.9836,E2 185.6297} C_DIS
LIN {X -14.4406,Y -116.8793,Z 129,A -100.8982,B 24.959,C -1.4808,E1 24.9797,E2 187.0325} C_DIS
LIN {X -17.296,Y -116.4911,Z 129,A -102.3012,B 24.959,C -1.481,E1 24.9758,E2 188.436} C_DIS
LIN {X -20.5495,Y -115.9596,Z 129,A -103.9763,B 24.959,C -1.4784,E1 24.9712,E2 190.119} C_DIS
LIN {X -23.7255,Y -115.3513,Z 129,A -105.4622,B 24.9588,C -1.4829,E1 24.9672,E2 191.5957} C_DIS
LIN {X -26.5556,Y -114.7328,Z 129,A -106.8735,B 24.9588,C -1.4835,E1 24.9633,E2 193.0075} C_DIS
LIN {X -29.3821,Y -114.0417,Z 129,A -108.3438,B 24.9588,C -1.4819,E1 24.9593,E2 194.4836} C_DIS
LIN {X -32.8085,Y -113.1058,Z 129,A -110.0402,B 24.9588,C -1.4844,E1 24.9548,E2 196.1768} C_DIS
LIN {X -35.5687,Y -112.2685,Z 129,A -111.5967,B 24.959,C -1.4787,E1 24.9506,E2 197.7496} C_DIS
LIN {X -39.0505,Y -111.103,Z 129,A -113.2187,B 24.9585,C -1.4875,E1 24.9463,E2 199.3538} C_DIS
LIN {X -41.6812,Y -110.1431,Z 129,A -114.6199,B 24.9585,C -1.4871,E1 24.9427,E2 200.7589} C_DIS
LIN {X -44.4438,Y -109.0576,Z 129,A -116.087,B 24.9585,C -1.4875,E1 24.9388,E2 202.2282} C_DIS
LIN {X -47.7299,Y -107.6624,Z 129,A -117.8677,B 24.9585,C -1.4875,E1 24.9343,E2 204.0133} C_DIS
LIN {X -50.3543,Y -106.4602,Z 129,A -119.1972,B 24.9583,C -1.4923,E1 24.9309,E2 205.3344} C_DIS
LIN {X -52.9465,Y -105.1951,Z 129,A -120.6051,B 24.9582,C -1.4939,E1 24.9274,E2 206.7424} C_DIS
LIN {X -55.9911,Y -103.6043,Z 129,A -122.3254,B 24.9582,C -1.494,E1 24.9232,E2 208.4671} C_DIS
LIN {X -58.652,Y -102.1213,Z 129,A -123.7671,B 24.958,C -1.4979,E1 24.9197,E2 209.9039} C_DIS
LIN {X -61.1344,Y -100.6549,Z 129,A -125.1937,B 24.958,C -1.4989,E1 24.9162,E2 211.3324} C_DIS
LIN {X -63.6552,Y -99.0799,Z 129,A -126.6059,B 24.9577,C -1.5026,E1 24.9129,E2 212.7403} C_DIS
LIN {X -65.9889,Y -97.5412,Z 129,A -128.0067,B 24.9577,C -1.5031,E1 24.9097,E2 214.1447} C_DIS
LIN {X -68.4036,Y -95.8632,Z 129,A -129.4228,B 24.9575,C -1.5061,E1 24.9064,E2 215.5584} C_DIS
LIN {X -70.7094,Y -94.1754,Z 129,A -130.8288,B 24.9575,C -1.5079,E1 24.9033,E2 216.9652} C_DIS
LIN {X -73.0441,Y -92.3763,Z 129,A -132.258,B 24.9572,C -1.5107,E1 24.9001,E2 218.3928} C_DIS
LIN {X -75.2728,Y -90.5694,Z 129,A -133.6631,B 24.9572,C -1.513,E1 24.8971,E2 219.798} C_DIS
LIN {X -77.4693,Y -88.6979,Z 129,A -135.114,B 24.9571,C -1.5137,E1 24.894,E2 221.2527} C_DIS
LIN {X -80.1577,Y -86.2791,Z 129,A -136.9762,B 24.9571,C -1.5129,E1 24.8902,E2 223.1243} C_DIS
LIN {X -82.4947,Y -84.0451,Z 129,A -138.4338,B 24.9566,C -1.5211,E1 24.8873,E2 224.5684} C_DIS
LIN {X -84.5571,Y -81.9696,Z 129,A -139.8346,B 24.9564,C -1.5252,E1 24.8845,E2 225.9656} C_DIS
LIN {X -86.5075,Y -79.9088,Z 129,A -141.2575,B 24.9564,C -1.5265,E1 24.8818,E2 227.3916} C_DIS
LIN {X -88.4797,Y -77.7192,Z 129,A -142.6632,B 24.9561,C -1.5309,E1 24.8792,E2 228.793} C_DIS
LIN {X -90.5097,Y -75.3447,Z 129,A -144.2311,B 24.956,C -1.5325,E1 24.8764,E2 230.3644} C_DIS
LIN {X -92.4098,Y -73.0016,Z 129,A -145.6803,B 24.9558,C -1.5368,E1 24.8738,E2 231.8101} C_DIS
LIN {X -94.371,Y -70.449,Z 129,A -147.2909,B 24.9556,C -1.5388,E1 24.8711,E2 233.4236} C_DIS
LIN {X -96.2828,Y -67.8156,Z 129,A -148.8521,B 24.9554,C -1.5437,E1 24.8686,E2 234.9809} C_DIS
LIN {X -97.9239,Y -65.4236,Z 129,A -150.4213,B 24.9555,C -1.5407,E1 24.8661,E2 236.5649} C_DIS
LIN {X -99.8565,Y -62.4299,Z 129,A -152.0301,B 24.955,C -1.5506,E1 24.8637,E2 238.1585} C_DIS
LIN {X -101.4701,Y -59.7718,Z 129,A -153.6286,B 24.955,C -1.551,E1 24.8614,E2 239.7641} C_DIS
LIN {X -103.1978,Y -56.7404,Z 129,A -155.2318,B 24.9544,C -1.5596,E1 24.8593,E2 241.3552} C_DIS
LIN {X -104.7185,Y -53.8791,Z 129,A -156.6484,B 24.9538,C -1.5707,E1 24.8574,E2 242.753} C_DIS
LIN {X -105.922,Y -51.4745,Z 129,A -158.0582,B 24.9538,C -1.5701,E1 24.8557,E2 244.1717} C_DIS
LIN {X -107.0735,Y -49.0368,Z 129,A -159.461,B 24.9538,C -1.5701,E1 24.854,E2 245.5822} C_DIS
LIN {X -108.2423,Y -46.3997,Z 129,A -160.8744,B 24.9536,C -1.5737,E1 24.8524,E2 246.9948} C_DIS
LIN {X -109.4656,Y -43.431,Z 129,A -162.3181,B 24.953,C -1.5833,E1 24.8509,E2 248.4238} C_DIS
LIN {X -110.3948,Y -41.0158,Z 129,A -163.7805,B 24.9533,C -1.5786,E1 24.8495,E2 249.9056} C_DIS
LIN {X -111.3644,Y -38.3052,Z 129,A -165.1255,B 24.9529,C -1.5851,E1 24.8482,E2 251.2427} C_DIS
LIN {X -112.2785,Y -35.5365,Z 129,A -166.5373,B 24.9527,C -1.5897,E1 24.847,E2 252.6517} C_DIS
LIN {X -113.1035,Y -32.8165,Z 129,A -167.9432,B 24.9525,C -1.593,E1 24.8459,E2 254.0579} C_DIS
LIN {X -113.8758,Y -30.027,Z 129,A -169.5362,B 24.9526,C -1.5897,E1 24.8447,E2 255.6679} C_DIS
LIN {X -114.7532,Y -26.4673,Z 129,A -171.1592,B 24.9519,C -1.6019,E1 24.8437,E2 257.2713} C_DIS
LIN {X -115.3521,Y -23.7215,Z 129,A -172.5521,B 24.9517,C -1.6052,E1 24.8429,E2 258.6647} C_DIS
LIN {X -115.8985,Y -20.8893,Z 129,A -173.9462,B 24.9514,C -1.61,E1 24.8422,E2 260.0555} C_DIS
LIN {X -116.3893,Y -17.954,Z 129,A -175.3837,B 24.9511,C -1.6151,E1 24.8415,E2 261.4895} C_DIS
LIN {X -116.7948,Y -15.0925,Z 129,A -176.8527,B 24.9511,C -1.617,E1 24.841,E2 262.9626} C_DIS
LIN {X -117.2016,Y -11.5371,Z 129,A -178.5719,B 24.9506,C -1.6234,E1 24.8405,E2 264.6767} C_DIS
LIN {X -117.4491,Y -8.6636,Z 129,A -179.9864,B 24.9504,C -1.6275,E1 24.8402,E2 266.09} C_DIS
LIN {X -117.626,Y -5.7845,Z 129,A 178.5048,B 24.9504,C -1.6278,E1 24.8399,E2 267.6074} C_DIS
LIN {X -117.74,Y -2.4928,Z 129,A 176.9162,B 24.95,C -1.6336,E1 24.8399,E2 269.1917} C_DIS
LIN {X -117.7651,Y 0.5257,Z 129,A 175.4621,B 24.9497,C -1.639,E1 24.8398,E2 270.6417} C_DIS
LIN {X -117.712,Y 3.5658,Z 129,A 173.9988,B 24.9493,C -1.6445,E1 24.8398,E2 272.1007} C_DIS
LIN {X -117.5844,Y 6.5361,Z 129,A 172.5209,B 24.9491,C -1.6479,E1 24.8401,E2 273.5793} C_DIS
LIN {X -117.3229,Y 10.2229,Z 129,A 170.7749,B 24.9486,C -1.6559,E1 24.8405,E2 275.3167} C_DIS
LIN {X -117.0503,Y 12.9836,Z 129,A 169.3924,B 24.9484,C -1.6589,E1 24.8409,E2 276.7003} C_DIS
LIN {X -116.697,Y 15.8476,Z 129,A 167.9772,B 24.9482,C -1.6631,E1 24.8414,E2 278.114} C_DIS
LIN {X -116.2739,Y 18.7005,Z 129,A 166.5642,B 24.9479,C -1.6672,E1 24.842,E2 279.5255} C_DIS
LIN {X -115.6856,Y 22.0387,Z 129,A 164.8562,B 24.9477,C -1.6702,E1 24.8428,E2 281.2365} C_DIS
LIN {X -115.0604,Y 25.0983,Z 129,A 163.3564,B 24.9474,C -1.6759,E1 24.8437,E2 282.7315} C_DIS
LIN {X -114.4137,Y 27.8983,Z 129,A 161.9481,B 24.9471,C -1.68,E1 24.8446,E2 284.1384} C_DIS
LIN {X -113.6751,Y 30.7701,Z 129,A 160.5334,B 24.9467,C -1.6858,E1 24.8456,E2 285.5476} C_DIS
LIN {X -112.9143,Y 33.4542,Z 129,A 159.1475,B 24.9465,C -1.6889,E1 24.8467,E2 286.9339} C_DIS
LIN {X -112.0357,Y 36.2881,Z 129,A 157.7139,B 24.9462,C -1.6939,E1 24.8479,E2 288.3639} C_DIS
LIN {X -111.1344,Y 38.9611,Z 129,A 156.3116,B 24.946,C -1.697,E1 24.8492,E2 289.7667} C_DIS
LIN {X -110.1469,Y 41.6711,Z 129,A 154.8791,B 24.9458,C -1.7002,E1 24.8506,E2 291.1998} C_DIS
LIN {X -108.9633,Y 44.6757,Z 129,A 153.2612,B 24.9456,C -1.7032,E1 24.8522,E2 292.8196} C_DIS
LIN {X -107.655,Y 47.7463,Z 129,A 151.5614,B 24.9456,C -1.705,E1 24.8541,E2 294.5244} C_DIS
LIN {X -106.4558,Y 50.3636,Z 129,A 150.2742,B 24.9449,C -1.7139,E1 24.8556,E2 295.7974} C_DIS
LIN {X -105.1925,Y 52.9515,Z 129,A 148.8625,B 24.9447,C -1.7177,E1 24.8574,E2 297.2077} C_DIS
LIN {X -103.8663,Y 55.5079,Z 129,A 147.4515,B 24.9445,C -1.7215,E1 24.8592,E2 298.6171} C_DIS
LIN {X -102.4781,Y 58.0305,Z 129,A 146.0418,B 24.9442,C -1.7253,E1 24.8611,E2 300.0253} C_DIS
LIN {X -101.0295,Y 60.5171,Z 129,A 144.6324,B 24.944,C -1.729,E1 24.8631,E2 301.4332} C_DIS
LIN {X -99.1988,Y 63.4701,Z 129,A 142.8958,B 24.9438,C -1.7319,E1 24.8657,E2 303.1715} C_DIS
LIN {X -97.5337,Y 65.9999,Z 129,A 141.4505,B 24.9434,C -1.7373,E1 24.8679,E2 304.6113} C_DIS
LIN {X -95.891,Y 68.3647,Z 129,A 140.0411,B 24.9432,C -1.7408,E1 24.8702,E2 306.0192} C_DIS
LIN {X -94.0871,Y 70.8269,Z 129,A 138.504,B 24.9431,C -1.7427,E1 24.8728,E2 307.5592} C_DIS
LIN {X -91.6795,Y 73.9173,Z 129,A 136.6328,B 24.9427,C -1.7493,E1 24.876,E2 309.4236} C_DIS
LIN {X -89.6627,Y 76.3506,Z 129,A 135.0752,B 24.9424,C -1.7525,E1 24.8788,E2 310.9807} C_DIS
LIN {X -87.7461,Y 78.5457,Z 129,A 133.6543,B 24.9422,C -1.756,E1 24.8814,E2 312.3996} C_DIS
LIN {X -85.7856,Y 80.6823,Z 129,A 132.2388,B 24.942,C -1.7594,E1 24.8841,E2 313.8132} C_DIS
LIN {X -83.7518,Y 82.7916,Z 129,A 130.8081,B 24.9418,C -1.7627,E1 24.8869,E2 315.2422} C_DIS
LIN {X -81.7136,Y 84.8039,Z 129,A 129.4068,B 24.9416,C -1.7658,E1 24.8897,E2 316.6421} C_DIS
LIN {X -79.6242,Y 86.7687,Z 129,A 127.9995,B 24.9414,C -1.7686,E1 24.8926,E2 318.0485} C_DIS
LIN {X -77.4646,Y 88.702,Z 129,A 126.5849,B 24.9412,C -1.7716,E1 24.8955,E2 319.4613} C_DIS
LIN {X -75.2132,Y 90.6189,Z 129,A 125.091,B 24.9412,C -1.7726,E1 24.8987,E2 320.9587} C_DIS
LIN {X -72.1803,Y 93.0536,Z 129,A 123.3896,B 24.9403,C -1.7847,E1 24.9024,E2 322.6376} C_DIS
LIN {X -70.158,Y 94.5895,Z 129,A 121.9966,B 24.9406,C -1.7807,E1 24.9055,E2 324.0453} C_DIS
LIN {X -67.8095,Y 96.2871,Z 129,A 120.5818,B 24.9404,C -1.7833,E1 24.9087,E2 325.4585} C_DIS
LIN {X -65.0911,Y 98.1431,Z 129,A 119.1002,B 24.9398,C -1.7916,E1 24.9121,E2 326.9254} C_DIS
LIN {X -62.9464,Y 99.5339,Z 129,A 117.7302,B 24.94,C -1.7887,E1 24.9154,E2 328.3068} C_DIS
LIN {X -60.4071,Y 101.0946,Z 129,A 116.324,B 24.9397,C -1.7932,E1 24.9187,E2 329.7065} C_DIS
LIN {X -58.0317,Y 102.4775,Z 129,A 114.9293,B 24.9397,C -1.7932,E1 24.9221,E2 331.1055} C_DIS
LIN {X -55.517,Y 103.8615,Z 129,A 113.3551,B 24.9401,C -1.7881,E1 24.926,E2 332.6962} C_DIS
LIN {X -52.9362,Y 105.2002,Z 129,A 112.1051,B 24.9394,C -1.7974,E1 24.9291,E2 333.9276} C_DIS
LIN {X -50.3443,Y 106.4649,Z 129,A 110.6972,B 24.9394,C -1.7994,E1 24.9326,E2 335.3342} C_DIS
LIN {X -47.7218,Y 107.666,Z 129,A 109.2147,B 24.9394,C -1.7982,E1 24.9364,E2 336.8233} C_DIS
LIN {X -44.6526,Y 108.9727,Z 129,A 107.5523,B 24.9394,C -1.7988,E1 24.9407,E2 338.4878} C_DIS
LIN {X -40.9273,Y 110.4271,Z 129,A 105.725,B 24.9388,C -1.8065,E1 24.9454,E2 340.3008} C_DIS
LIN {X -38.2721,Y 111.3756,Z 129,A 104.3453,B 24.9388,C -1.8079,E1 24.9491,E2 341.6799} C_DIS
LIN {X -35.0391,Y 112.4327,Z 129,A 102.9061,B 24.938,C -1.8192,E1 24.9528,E2 343.0949} C_DIS
LIN {X -32.7883,Y 113.1117,Z 129,A 101.5286,B 24.9386,C -1.8103,E1 24.9566,E2 344.4957} C_DIS
LIN {X -30.0085,Y 113.8807,Z 129,A 100.1223,B 24.9385,C -1.8117,E1 24.9604,E2 345.9009} C_DIS
LIN {X -27.2105,Y 114.5815,Z 129,A 98.5391,B 24.9389,C -1.8052,E1 24.9647,E2 347.5016} C_DIS
LIN {X -23.7029,Y 115.3559,Z 129,A 96.9457,B 24.9384,C -1.8135,E1 24.969,E2 349.0774} C_DIS
LIN {X -20.598,Y 115.9509,Z 129,A 95.368,B 24.9384,C -1.813,E1 24.9733,E2 350.6579} C_DIS
LIN {X -17.0053,Y 116.5326,Z 129,A 93.7713,B 24.9378,C -1.8217,E1 24.9777,E2 352.2352} C_DIS
LIN {X -14.4188,Y 116.8821,Z 129,A 92.3731,B 24.9381,C -1.8169,E1 24.9816,E2 353.646} C_DIS
LIN {X -11.5361,Y 117.2017,Z 129,A 90.9588,B 24.9381,C -1.8175,E1 24.9855,E2 355.0596} C_DIS
LIN {X -8.6461,Y 117.4502,Z 129,A 89.5545,B 24.9381,C -1.8185,E1 24.9894,E2 356.4623} C_DIS
LIN {X -5.7698,Y 117.6267,Z 129,A 88.1513,B 24.938,C -1.8189,E1 24.9933,E2 357.8647} C_DIS
LIN {X -2.8895,Y 117.7327,Z 129,A 86.7317,B 24.938,C -1.8186,E1 24.9973,E2 359.2854} C_DIS
LIN {X 0.0289,Y 117.768,Z 129,A 85.3281,B 24.938,C -1.8196,E1 25.0012,E2 360.6866} C_DIS
LIN {X 2.9086,Y 117.7321,Z 129,A 83.9263,B 24.938,C -1.8198,E1 25.0051,E2 362.0878} C_DIS
LIN {X 5.8465,Y 117.6225,Z 129,A 82.5212,B 24.9378,C -1.821,E1 25.009,E2 363.4896} C_DIS
LIN {X 8.6641,Y 117.449,Z 129,A 81.0831,B 24.938,C -1.8181,E1 25.0131,E2 364.934} C_DIS
LIN {X 11.565,Y 117.1988,Z 129,A 79.7058,B 24.938,C -1.8197,E1 25.0169,E2 366.3067} C_DIS
LIN {X 14.4301,Y 116.8807,Z 129,A 78.3036,B 24.938,C -1.8194,E1 25.0208,E2 367.7084} C_DIS
LIN {X 17.2871,Y 116.4924,Z 129,A 76.9017,B 24.938,C -1.8191,E1 25.0246,E2 369.1099} C_DIS
LIN {X 20.1341,Y 116.0343,Z 129,A 75.4982,B 24.938,C -1.8186,E1 25.0285,E2 370.5132} C_DIS
LIN {X 22.969,Y 115.5065,Z 129,A 74.0951,B 24.938,C -1.818,E1 25.0324,E2 371.9161} C_DIS
LIN {X 26.3382,Y 114.783,Z 129,A 72.3873,B 24.9382,C -1.8157,E1 25.037,E2 373.6268} C_DIS
LIN {X 29.3662,Y 114.0458,Z 129,A 70.9079,B 24.9382,C -1.8165,E1 25.041,E2 375.1023} C_DIS
LIN {X 32.8016,Y 113.1079,Z 129,A 68.9627,B 24.9389,C -1.8057,E1 25.0463,E2 377.0698} C_DIS
LIN {X 36.8547,Y 111.8523,Z 129,A 67.106,B 24.9384,C -1.8134,E1 25.0512,E2 378.9049} C_DIS
LIN {X 39.6866,Y 110.8796,Z 129,A 65.6648,B 24.9384,C -1.8128,E1 25.055,E2 380.3446} C_DIS
LIN {X 42.3855,Y 109.8763,Z 129,A 64.2613,B 24.9385,C -1.8113,E1 25.0587,E2 381.7486} C_DIS
LIN {X 45.0734,Y 108.8013,Z 129,A 62.8601,B 24.9385,C -1.8102,E1 25.0623,E2 383.1493} C_DIS
LIN {X 47.7253,Y 107.6644,Z 129,A 61.4592,B 24.9387,C -1.8087,E1 25.0659,E2 384.5502} C_DIS
LIN {X 50.3478,Y 106.4633,Z 129,A 60.0589,B 24.9387,C -1.8072,E1 25.0694,E2 385.9506} C_DIS
LIN {X 53.4333,Y 104.9463,Z 129,A 58.3941,B 24.9389,C -1.8054,E1 25.0736,E2 387.615} C_DIS
LIN {X 56.1315,Y 103.5281,Z 129,A 56.894,B 24.9391,C -1.8026,E1 25.0773,E2 389.1175} C_DIS
LIN {X 58.6477,Y 102.1238,Z 129,A 55.5152,B 24.9391,C -1.8017,E1 25.0806,E2 390.4945} C_DIS
LIN {X 61.1294,Y 100.6579,Z 129,A 54.098,B 24.9393,C -1.7989,E1 25.084,E2 391.9139} C_DIS
LIN {X 63.6494,Y 99.0836,Z 129,A 52.696,B 24.9393,C -1.7986,E1 25.0873,E2 393.312} C_DIS
LIN {X 65.9821,Y 97.5458,Z 129,A 51.3221,B 24.9396,C -1.7957,E1 25.0905,E2 394.6883} C_DIS
LIN {X 68.3494,Y 95.902,Z 129,A 49.9075,B 24.9398,C -1.7927,E1 25.0938,E2 396.105} C_DIS
LIN {X 70.7085,Y 94.1761,Z 129,A 48.4988,B 24.9398,C -1.7908,E1 25.0969,E2 397.5132} C_DIS
LIN {X 73.0267,Y 92.39,Z 129,A 47.0897,B 24.94,C -1.7888,E1 25.1,E2 398.9217} C_DIS
LIN {X 75.2685,Y 90.573,Z 129,A 45.6524,B 24.9403,C -1.7846,E1 25.1031,E2 400.3635} C_DIS
LIN {X 78.045,Y 88.1945,Z 129,A 43.8078,B 24.9408,C -1.7779,E1 25.107,E2 402.2166} C_DIS
LIN {X 80.4141,Y 86.0379,Z 129,A 42.3496,B 24.9407,C -1.7794,E1 25.11,E2 403.6653} C_DIS
LIN {X 82.4897,Y 84.05,Z 129,A 40.964,B 24.9408,C -1.777,E1 25.1128,E2 405.0508} C_DIS
LIN {X 84.5633,Y 81.9632,Z 129,A 39.5669,B 24.9409,C -1.7755,E1 25.1155,E2 406.4456} C_DIS
LIN {X 86.5158,Y 79.8998,Z 129,A 38.1624,B 24.9412,C -1.7713,E1 25.1182,E2 407.8538} C_DIS
LIN {X 88.5878,Y 77.5955,Z 129,A 36.6345,B 24.9415,C -1.7669,E1 25.121,E2 409.3853} C_DIS
LIN {X 90.5724,Y 75.2692,Z 129,A 35.1958,B 24.9415,C -1.7657,E1 25.1236,E2 410.8202} C_DIS
LIN {X 92.3894,Y 73.0275,Z 129,A 33.6984,B 24.9421,C -1.7579,E1 25.1263,E2 412.3291} C_DIS
LIN {X 94.6042,Y 70.1381,Z 129,A 32.0387,B 24.9421,C -1.7587,E1 25.129,E2 413.979} C_DIS
LIN {X 96.2923,Y 67.802,Z 129,A 30.6439,B 24.9422,C -1.7555,E1 25.1313,E2 415.3746} C_DIS
LIN {X 98.1317,Y 65.1083,Z 129,A 29.2316,B 24.942,C -1.7597,E1 25.1335,E2 416.7701} C_DIS
LIN {X 99.4952,Y 63.0083,Z 129,A 27.8527,B 24.9427,C -1.7488,E1 25.1356,E2 418.1677} C_DIS
LIN {X 101.0076,Y 60.554,Z 129,A 26.4582,B 24.9429,C -1.7454,E1 25.1376,E2 419.563} C_DIS
LIN {X 102.6365,Y 57.747,Z 129,A 25.039,B 24.9427,C -1.7487,E1 25.1396,E2 420.9671} C_DIS
LIN {X 104.031,Y 55.195,Z 129,A 23.4499,B 24.9435,C -1.7365,E1 25.1417,E2 422.5767} C_DIS
LIN {X 105.1973,Y 52.9419,Z 129,A 22.2563,B 24.9435,C -1.7349,E1 25.1432,E2 423.7677} C_DIS
LIN {X 106.4624,Y 50.3497,Z 129,A 20.8615,B 24.9438,C -1.7313,E1 25.1449,E2 425.1635} C_DIS
LIN {X 107.8467,Y 47.3074,Z 129,A 19.437,B 24.9435,C -1.7362,E1 25.1465,E2 426.5686} C_DIS
LIN {X 108.8051,Y 45.0642,Z 129,A 18.0663,B 24.9443,C -1.724,E1 25.148,E2 427.9607} C_DIS
LIN {X 110.3674,Y 41.0887,Z 129,A 15.9508,B 24.9448,C -1.716,E1 25.1502,E2 430.0832} C_DIS
LIN {X 111.3758,Y 38.2715,Z 129,A 14.5675,B 24.9448,C -1.7151,E1 25.1514,E2 431.461} C_DIS
LIN {X 112.2708,Y 35.561,Z 129,A 13.1746,B 24.9452,C -1.7106,E1 25.1526,E2 432.8565} C_DIS
LIN {X 113.1081,Y 32.8007,Z 129,A 11.7792,B 24.9454,C -1.7067,E1 25.1537,E2 434.2533} C_DIS
LIN {X 113.8778,Y 30.0197,Z 129,A 10.2666,B 24.946,C -1.6971,E1 25.1549,E2 435.7796} C_DIS
LIN {X 114.6777,Y 26.7944,Z 129,A 8.7619,B 24.946,C -1.6975,E1 25.1558,E2 437.2749} C_DIS
LIN {X 115.3519,Y 23.7224,Z 129,A 7.24,B 24.9463,C -1.693,E1 25.1567,E2 438.7983} C_DIS
LIN {X 115.8981,Y 20.8911,Z 129,A 5.8661,B 24.9465,C -1.69,E1 25.1574,E2 440.1714} C_DIS
Enddeposition()
END
